// TwinCAT 3 PLC project plc_kfe_vac
// Title: plc_kfe_vac
// Company: SLAC
// ProjectVersion: 0.0.0
// ProgramVersion: 3.1.4022.4
// libraries:
//   LCLS General, * (SLAC)
//   LCLS Vacuum, * (SLAC - LCLS)
//   PMPS, * (SLAC - LCLS)
//   Tc2_Standard, * (Beckhoff Automation GmbH)
//   Tc2_System, * (Beckhoff Automation GmbH)
//   Tc2_Utilities, * (Beckhoff Automation GmbH)
//   Tc3_Module, * (Beckhoff Automation GmbH)
// project tree:
//   DUTs/ ST_EXT_GCC.TcDUT, ST_EXT_ILK.TcDUT
//   / FSV_task.TcTTO, PlcTask.TcTTO
//   GVLs/ GVL_SXR_VAC.TcGVL, GVL_VAC_INTF.TcGVL, GVL_Variables.TcGVL, GVL_VFS.TcGVL
//   POUs/ FB_EXT_TREATY_GAUGE.TcPOU, FB_EXT_TREATY_VGC.TcPOU, FB_EXT_ILK.TcPOU, MAIN.TcPOU, PRG_DIAGNOSTIC.TcPOU, PRG_PMPS.TcPOU, PRG_SXR_VAC.TcPOU, PRG_VAC_INTF.TcPOU, PRG_VFS.TcPOU
// real-time tasks:
//   TASK PlcTask: cycle T#10ms, priority 20, ADS port 350
//   TASK SimTask: cycle T#10ms, priority 21, ADS port 351
//   TASK FSV_task: cycle T#1ms, priority 13, ADS port 352
// I/O:
//   DEVICE Device 1 (EtherCAT), AmsNetId 172.21.92.61.4.1
//     =+-EK1200_00_00 [EK1200-5000 EtherCAT Power supply (2A E-Bus)]
//       =+-ES3064_00_01 [EL3064 4Ch. Ana. Input 0-10V]
//       =+-ES1004_00_02 [EL1004 4Ch. Dig. Input 24V, 3ms]
//       =+-EL2794_00_03 [EL2794 4Ch. Dig. Output 24V AC/DC, 2A, short-circuit-proof]
//       =+-ES3064_00_04 [EL3064 4Ch. Ana. Input 0-10V]
//       =+-ES1004_00_05 [EL1004 4Ch. Dig. Input 24V, 3ms]
//       =+-EL2794_00_06 [EL2794 4Ch. Dig. Output 24V AC/DC, 2A, short-circuit-proof]
//       =+-EL9410_00_07 [EL9410 E-Bus Power Supplier  (Diagnostics)]
//       =+-ES3064_00_08 [EL3064 4Ch. Ana. Input 0-10V]
//       =+-ES1004_00_09 [EL1004 4Ch. Dig. Input 24V, 3ms]
//       =+-EL2794_00_10 [EL2794 4Ch. Dig. Output 24V AC/DC, 2A, short-circuit-proof]
//       =+-ES3064_00_11 [EL3064 4Ch. Ana. Input 0-10V]
//       =+-ES1004_00_12 [EL1004 4Ch. Dig. Input 24V, 3ms]
//       =+-EL2794_00_13 [EL2794 4Ch. Dig. Output 24V AC/DC, 2A, short-circuit-proof]
//       Term 81 (EL6070) [EL6070 1Ch. Licensing-Terminal]
//       =+-EK1110_00_14 [EK1110 EtherCAT extension]
//     =+-EK1100_01_00 [EK1100 EtherCAT Coupler (2A E-Bus)]
//       =+-ES3068_01_01 [EL3068 8Ch. Ana. Input 0-10V]
//       =+-EL2798_01_02 [EL2798 8Ch. Dig. Output 24V AC/DC, 2A, potential-free]
//       =+-ES9187_01_03 [EL9187 Potential Connection, 8 x Ground]
//       =+-ES3068_01_04 [EL3068 8Ch. Ana. Input 0-10V]
//       =+-ES3068_01_05 [EL3068 8Ch. Ana. Input 0-10V]
//       =+-EL2798_01_06 [EL2798 8Ch. Dig. Output 24V AC/DC, 2A, potential-free]
//       =+-ES9187_01_07 [EL9187 Potential Connection, 8 x Ground]
//       =+-ES3068_01_08 [EL3068 8Ch. Ana. Input 0-10V]
//       =+-EL9410_01_09 [EL9410 E-Bus Power Supplier  (Diagnostics)]
//       =+-EL2022_01_10 [EL2022 2Ch. Dig. Output 24V, 2A] (disabled)
//       PMPS_FFO (EL2202) [EL2202 2Ch. Dig. Output 24V, 0.5A]
//       PMPS_PRE [EL6692 EtherCAT Bridge terminal (Primary)]
//       =+-EL6695_01_11 [EL6695 EtherCAT Bridge terminal (Primary)] (disabled)
//       Term 73 (EK1122) [EK1122 2 port EtherCAT junction]
//       =+-EL6695_01_12 [EL6695 EtherCAT Bridge terminal (Primary)] (disabled)
//       Term 74 (EK1122) [EK1122 2 port EtherCAT junction]
//       =+-EL6695_01_13 [EL6695 EtherCAT Bridge terminal (Primary)] (disabled)
//       Term 75 (EK1122) [EK1122 2 port EtherCAT junction]
//       =+-EL6695_01_14 [EL6695 EtherCAT Bridge terminal (Primary)] (disabled)
//       Term 76 (EL9011) [EL9011 End Terminal]
//     =+-EK1100_02_00 [EK1100 EtherCAT Coupler (2A E-Bus)]
//       =+-EL3064_02_01 [EL3064 4Ch. Ana. Input 0-10V]
//       =+-EL9070_02_02 [EL9070 Shield terminal]
//       =+-ES1008_02_03 [EL1008 8Ch. Dig. Input 24V, 3ms]
//       =+-ES9184_02_04 [EL9184 Potential Connection, 8 x 24V, 8 x Ground]
//       =+-ES2008_02_05 [EL2008 8Ch. Dig. Output 24V, 0.5A]
//       =+-EL2798_02_06 [EL2798 8Ch. Dig. Output 24V AC/DC, 2A, potential-free]
//       =+-EL3064_02_07 [EL3064 4Ch. Ana. Input 0-10V]
//       =+-EL2794_02_08 [EL2794 4Ch. Dig. Output 24V AC/DC, 2A, short-circuit-proof]
//       =+-EL1004_02_09 [EL1004 4Ch. Dig. Input 24V, 3ms]
//       =+-EL9505_02_10 [EL9505 Power supply terminal 5V]
//       =+-EL1124_02_11 [EL1124 4Ch. Dig. Input 5V, 10µs, Sensor Power]
//       =+-EL9011_02_12 [EL9011 End Terminal]
//     =+-EK1100_03_00 [EK1100 EtherCAT Coupler (2A E-Bus)]
//       =+-ES1004_03_01 [EL1004 4Ch. Dig. Input 24V, 3ms]
//       =+-ES2004_03_02 [EL2004 4Ch. Dig. Output 24V, 0.5A]
//       =+-ES2004_03_03 [EL2004 4Ch. Dig. Output 24V, 0.5A]
//       =+-EL1004_03_04 [EL1004 4Ch. Dig. Input 24V, 3ms]
//       =+-EL3064_03_05 [EL3064 4Ch. Ana. Input 0-10V]
//       =+-EL9070_03_06 [EL9070 Shield terminal]
//       =+-ES1008_03_07 [EL1008 8Ch. Dig. Input 24V, 3ms]
//       =+-ES9184_03_08 [EL9184 Potential Connection, 8 x 24V, 8 x Ground]
//       =+-ES2008_03_09 [EL2008 8Ch. Dig. Output 24V, 0.5A]
//       =+-EL2798_03_10 [EL2798 8Ch. Dig. Output 24V AC/DC, 2A, potential-free]
//       =+-EL9011_03_11 [EL9011 End Terminal]
//     =+-EP2338_04_00 [EP2338-0002 8 Ch. Dig. Input/Output 24V, 0,5A, M12]
//     =+-EP2338_05_00 [EP2338-0002 8 Ch. Dig. Input/Output 24V, 0,5A, M12]
//     =+-EK1100_05_01 [EK1100 EtherCAT Coupler (2A E-Bus)]
//       =+-ES1004_05_02 [EL1004 4Ch. Dig. Input 24V, 3ms]
//       =+-ES2202_05_03 [EL2202 2Ch. Dig. Output 24V, 0.5A]
//       =+-ES2202_05_04 [EL2202 2Ch. Dig. Output 24V, 0.5A]
//       Term 55 (EL9011) [EL9011 End Terminal]
//     =+-EP2338_06_00 [EP2338-0002 8 Ch. Dig. Input/Output 24V, 0,5A, M12]
//     =+-EP2338_07_00 [EP2338-0002 8 Ch. Dig. Input/Output 24V, 0,5A, M12]
//     =+-EP3174_07_01 [EP3174-0002 4Ch. Ana. Input +/-10V, 0-10V, 0/4-20mA configurable]
//     =+-EP2624_07_02 [EP2624-0002 4Ch. Relay Output, NO (125V AC / 30V DC)]
//     =+-EP2338_08_00 [EP2338-0002 8 Ch. Dig. Input/Output 24V, 0,5A, M12]
//     =+-EP3174_08_01 [EP3174-0002 4Ch. Ana. Input +/-10V, 0-10V, 0/4-20mA configurable]
//     =+-EP2624_08_02 [EP2624-0002 4Ch. Relay Output, NO (125V AC / 30V DC)]
//     =+-EP3174_09_00 [EP3174-0002 4Ch. Ana. Input +/-10V, 0-10V, 0/4-20mA configurable]
//     =+-EP2624_09_01 [EP2624-0002 4Ch. Relay Output, NO (125V AC / 30V DC)]
//     =+-EP2338_09_02 [EP2338-0002 8 Ch. Dig. Input/Output 24V, 0,5A, M12]
//     =+-EP2338_09_03 [EP2338-0002 8 Ch. Dig. Input/Output 24V, 0,5A, M12]
//     =+-EP3174_10_00 [EP3174-0002 4Ch. Ana. Input +/-10V, 0-10V, 0/4-20mA configurable]
//     =+-EP2624_10_01 [EP2624-0002 4Ch. Relay Output, NO (125V AC / 30V DC)]
//     =+-EP2338_10_02 [EP2338-0002 8 Ch. Dig. Input/Output 24V, 0,5A, M12]
//   DEVICE SimDevice 2 (EtherCAT Simulation) (disabled), AmsNetId 10.0.1.49.3.1
//     =+-ES3064_00_01 // EL3064-0000-0020
//     =+-ES1004_00_02 // EL1004-0000-0019
//     =+-EL2794_00_03 // EL2794-0000-0016
//     =+-ES3064_00_04 // EL3064-0000-0020
//     =+-ES1004_00_05 // EL1004-0000-0019
//     =+-EL2794_00_06 // EL2794-0000-0016
//     =+-EL9410_00_07 // EL9410-0000-0017
//     =+-ES3064_00_08 // EL3064-0000-0020
//     =+-ES1004_00_09 // EL1004-0000-0019
//     =+-EL2794_00_10 // EL2794-0000-0016
//     =+-ES3064_00_11 // EL3064-0000-0020
//     =+-ES1004_00_12 // EL1004-0000-0019
//     =+-EL2794_00_13 // EL2794-0000-0016
//     =+-EK1110_00_14 // EK1110-0000-0017
//     =+-EK1100_01_00 // EK1100-0000-0018
//     =+-ES3068_01_01 // EL3068-0000-0020
//     =+-EL2798_01_02 // EL2798-0000-0018
//     =+-ES3068_01_04 // EL3068-0000-0020
//     =+-ES3068_01_05 // EL3068-0000-0020
//     =+-EL2798_01_06 // EL2798-0000-0018
//     =+-ES3068_01_08 // EL3068-0000-0020
//     =+-EL9410_01_09 // EL9410-0000-0017
//     =+-EL2202_01_10 // EL2022-0000-0018
//     =+-EL6695_01_11 // EL6695-0000-0005
//     =+-EL6695_01_12 // EL6695-0000-0005
//     =+-EL6695_01_13 // EL6695-0000-0005
//     =+-EL6695_01_14 // EL6695-0000-0005
//     =+-EK1100_02_00 // EK1100-0000-0018
//     =+-EL3064_02_01 // EL3064-0000-0020
//     =+-ES1008_02_03 // EL1008-0000-0018
//     =+-ES2008_02_05 // EL2008-0000-0018
//     =+-EL2798_02_06 // EL2798-0000-0018
//     =+-EK1100_03_00 // EK1100-0000-0018
//     =+-ES1004_03_01 // EL1004-0000-0019
//     =+-ES2004_03_02 // EL2004-0000-0018
//     =+-ES2004_03_03 // EL2004-0000-0018
//     =+-ES1004_03_04 // EL1008-0000-0018
//     =+-EL3064_03_05 // EL3064-0000-0020
//     =+-ES1008_03_07 // EL1008-0000-0018
//     =+-ES2008_03_09 // EL2008-0000-0018
//     =+-EL2798_03_10 // EL2798-0000-0018
//     =+-EP2338_04_00 // EP2338-0002-0023
//     =+-EP2338_05_00 // EP2338-0002-0023
//     =+-EK1100_05_01 // EK1100-0000-0018
//     =+-ES1004_05_02 // EL1004-0000-0019
//     =+-ES2202_05_03 // EL2202-0000-0019
//     =+-ES2202_05_04 // EL2202-0000-0019
//     =+-ES9505_05_05 // EL9505-0000-0018
//     =+-ES1124_05_06 // EL1124-0000-0018
//     =+-EP2338_06_00 // EP2338-0002-0023
//     =+-EP2338_07_00 // EP2338-0002-0023
//     =+-EP3174_07_01 // EP3174-0002-0023
//     =+-EP2624_07_02 // EP2624-0002-0019
//     =+-EP2338_08_00 // EP2338-0002-0023
//     =+-EP3174_08_01 // EP3174-0002-0023
//     =+-EP2624_08_02 // EP2624-0002-0019
//     =+-EP3174_09_00 // EP3174-0002-0023
//     =+-EP2624_09_01 // EP2624-0002-0019
//     =+-EP2338_09_02 // EP2338-0002-0023
//     =+-EP2338_09_03 // EP2338-0002-0023
//     =+-EP3174_10_00 // EP3174-0002-0023
//     =+-EP2624_10_01 // EP2624-0002-0019
//     =+-EP2338_10_02 // EP2338-0002-0023
//     =+-EP3174_11_00 // EP3174-0002-0023
//     =+-EP2624_11_01 // EP2624-0002-0019
//     =+-EP2338_11_02 // EP2338-0002-0023
//     =+-EK1100_11_03 // EK1100-0000-0018
//     =+-ES1004_11_04 // EL1004-0000-0019
//     =+-ES2202_11_05 // EL2202-0000-0019
//     =+-ES2202_11_06 // EL2202-0000-0019
//     =+-ES9505_11_07 // EL9505-0000-0018
//     =+-ES1124_11_08 // EL1124-0000-0018
//     =+-EP3174_12_00 // EP3174-0002-0023
//     =+-EP2624_12_01 // EP2624-0002-0019
//     =+-EP3174_13_00 // EP3174-0002-0023
//     =+-EP2624_13_01 // EP2624-0002-0019
//     =+-EP2338_14_00 // EP2338-0002-0023
//     =+-EP3174_14_01 // EP3174-0002-0023
//     =+-EP2624_14_02 // EP2624-0002-0019
//     =+-EK1100_15_00 // EK1100-0000-0018
//     =+-ES3064_15_01 // EL3064-0000-0020
//     =+-ES1004_15_02 // EL1004-0000-0019
//     =+-EL2794_15_03 // EL2794-0000-0016
//     =+-ES3064_15_04 // EL3064-0000-0020
//     =+-ES1004_15_05 // EL1004-0000-0019
//     =+-EL2794_15_06 // EL2794-0000-0016
// variable links:
//   plc_kfe_vac/plc_kfe_vac Instance <-> Device 1 (EtherCAT)
//     PlcTask Inputs/GVL_Variables.fbEcatDiagWrapper.arrEcMasterNetId <-> InfoData/AmsNetId
//     PlcTask Inputs/GVL_Variables.fbEcatDiagWrapper.nEcMasterDevState <-> Inputs/DevState
//     PlcTask Inputs/GVL_Variables.fbEcatDiagWrapper.nEcMasterDeviceId <-> InfoData/DevId
//     PlcTask Inputs/GVL_Variables.fbEcatDiagWrapper.nEcMasterSlaveCount <-> Inputs/SlaveCount
//     PlcTask Inputs/GVL_Variables.fbEcatDiagWrapper.nEcMasterSlaveCountCfg <-> InfoData/CfgSlaveCount
//     PlcTask Inputs/GVL_Variables.fbEcatDiagWrapper.wFrmXWcState <-> Inputs/Frm1WcState
//   plc_kfe_vac/plc_kfe_vac Instance <-> Device 1 (EtherCAT)/=+-EK1100_01_00/=+-EL2798_01_02
//     PlcTask Outputs/GVL_SXR_VAC.fb_IM1K0_XTES_GCC_1.q_xHV_DIS <-> Channel 2/GVL_SXR_VAC.fb_IM1K0_XTES_GCC_1.q_xHV_DIS
//     PlcTask Outputs/GVL_SXR_VAC.fb_PCPM3B_GFS_1.q_xHV_DIS <-> Channel 5/GVL_SXR_VAC.fb_PCPM3B_GFS_1.q_xHV_DIS
//     PlcTask Outputs/GVL_SXR_VAC.fb_RTDSK0_GCC_1.q_xHV_DIS <-> Channel 1/GVL_SXR_VAC.fb_RTDSK0_GCC_1.q_xHV_DIS
//     PlcTask Outputs/GVL_SXR_VAC.fb_SL1K0_POWER_GCC_1.q_xHV_DIS <-> Channel 4/GVL_SXR_VAC.fb_SL1K0_POWER_GCC_1.q_xHV_DIS
//   plc_kfe_vac/plc_kfe_vac Instance <-> Device 1 (EtherCAT)/=+-EK1100_01_00/=+-EL2798_01_06
//     PlcTask Outputs/GVL_SXR_VAC.fb_PA1K0_GCC_1.q_xHV_DIS <-> Channel 4/GVL_SXR_VAC.fb_PA1K0_GCC_1.q_xHV_DIS
//     PlcTask Outputs/GVL_SXR_VAC.fb_TV2K0_GCC_1.q_xHV_DIS <-> Channel 1/GVL_SXR_VAC.fb_TV2K0_GCC_1.q_xHV_DIS
//     PlcTask Outputs/GVL_SXR_VAC.fb_TV2K0_GCC_2.q_xHV_DIS <-> Channel 2/GVL_SXR_VAC.fb_TV2K0_GCC_2.q_xHV_DIS
//   plc_kfe_vac/plc_kfe_vac Instance <-> Device 1 (EtherCAT)/=+-EK1100_01_00/=+-ES3068_01_01
//     PlcTask Inputs/GVL_SXR_VAC.fb_IM1K0_XTES_GCC_1.i_iPRESS_R <-> AI Standard Channel 3/GVL_SXR_VAC.fb_IM1K0_XTES_GCC_1.i_iPRESS_R
//     PlcTask Inputs/GVL_SXR_VAC.fb_IM1K0_XTES_GPI_1.i_iPRESS_R <-> AI Standard Channel 6/GVL_SXR_VAC.fb_IM1K0_XTES_GPI_1.i_iPRESS_R
//     PlcTask Inputs/GVL_SXR_VAC.fb_RTDSK0_GCC_1.i_iPRESS_R <-> AI Standard Channel 1/GVL_SXR_VAC.fb_RTDSK0_GCC_1.i_iPRESS_R
//     PlcTask Inputs/GVL_SXR_VAC.fb_RTDSK0_GPI_1.i_iPRESS_R <-> AI Standard Channel 5/GVL_SXR_VAC.fb_RTDSK0_GPI_1.i_iPRESS_R
//   plc_kfe_vac/plc_kfe_vac Instance <-> Device 1 (EtherCAT)/=+-EK1100_01_00/=+-ES3068_01_04
//     PlcTask Inputs/GVL_SXR_VAC.fb_PCPM3B_GFS_1.i_iPRESS_R <-> AI Standard Channel 3/GVL_SXR_VAC.fb_PCPM3B_GFS_1.i_iPRESS_R
//     PlcTask Inputs/GVL_SXR_VAC.fb_SL1K0_POWER_GCC_1.i_iPRESS_R <-> AI Standard Channel 1/GVL_SXR_VAC.fb_SL1K0_POWER_GCC_1.i_iPRESS_R
//     PlcTask Inputs/GVL_SXR_VAC.fb_SL1K0_POWER_GPI_1.i_iPRESS_R <-> AI Standard Channel 5/GVL_SXR_VAC.fb_SL1K0_POWER_GPI_1.i_iPRESS_R
//   plc_kfe_vac/plc_kfe_vac Instance <-> Device 1 (EtherCAT)/=+-EK1100_01_00/=+-ES3068_01_05
//     PlcTask Inputs/GVL_SXR_VAC.fb_TV2K0_GCC_1.i_iPRESS_R <-> AI Standard Channel 1/GVL_SXR_VAC.fb_TV2K0_GCC_1.i_iPRESS_R
//     PlcTask Inputs/GVL_SXR_VAC.fb_TV2K0_GCC_2.i_iPRESS_R <-> AI Standard Channel 3/GVL_SXR_VAC.fb_TV2K0_GCC_2.i_iPRESS_R
//     PlcTask Inputs/GVL_SXR_VAC.fb_TV2K0_GPI_1.i_iPRESS_R <-> AI Standard Channel 5/GVL_SXR_VAC.fb_TV2K0_GPI_1.i_iPRESS_R
//     PlcTask Inputs/GVL_SXR_VAC.fb_TV2K0_GPI_2.i_iPRESS_R <-> AI Standard Channel 6/GVL_SXR_VAC.fb_TV2K0_GPI_2.i_iPRESS_R
//   plc_kfe_vac/plc_kfe_vac Instance <-> Device 1 (EtherCAT)/=+-EK1100_01_00/=+-ES3068_01_08
//     PlcTask Inputs/GVL_SXR_VAC.fb_PA1K0_GCC_1.i_iPRESS_R <-> AI Standard Channel 1/GVL_SXR_VAC.fb_PA1K0_GCC_1.i_iPRESS_R
//     PlcTask Inputs/GVL_SXR_VAC.fb_PA1K0_GPI_1.i_iPRESS_R <-> AI Standard Channel 5/GVL_SXR_VAC.fb_PA1K0_GPI_1.i_iPRESS_R
//   plc_kfe_vac/plc_kfe_vac Instance <-> Device 1 (EtherCAT)/=+-EK1100_01_00/PMPS_FFO (EL2202)
//     FSV_task Outputs/GVL_Variables.g_FastFaultOutput2.q_xFastFaultOut <-> Channel 2/Output
//     PlcTask Outputs/GVL_Variables.g_FastFaultOutputAll.q_xFastFaultOut <-> Channel 1/Output
//   plc_kfe_vac/plc_kfe_vac Instance <-> Device 1 (EtherCAT)/=+-EK1100_01_00/PMPS_PRE
//     PlcTask Inputs/PRG_PMPS.fbArbiterIO.i_stCurrentBP <-> IO Inputs/CurrentBP
//     PlcTask Inputs/PRG_PMPS.fbArbiterIO.xTxPDO_state <-> SYNC Inputs/TxPDO state
//     PlcTask Inputs/PRG_PMPS.fbArbiterIO.xTxPDO_toggle <-> SYNC Inputs/TxPDO toggle
//     PlcTask Outputs/PRG_PMPS.fbArbiterIO.q_stRequestedBP <-> IO Outputs/RequestedBP
//   plc_kfe_vac/plc_kfe_vac Instance <-> Device 1 (EtherCAT)/=+-EK1100_02_00/=+-EL1004_02_09
//     PlcTask Inputs/GVL_SXR_VAC.fb_SL1K0_PIP_1.i_xSP_DI <-> Channel 1/Input
//   plc_kfe_vac/plc_kfe_vac Instance <-> Device 1 (EtherCAT)/=+-EK1100_02_00/=+-EL1124_02_11
//     FSV_task Inputs/GVL_VFS.fb_TV2K0_VFS_1.i_xTrigger <-> Channel 1/GVL_SXR_VAC_FS_DEVICES.fb_TV2K0_VFS_1.i_xTrigger
//   plc_kfe_vac/plc_kfe_vac Instance <-> Device 1 (EtherCAT)/=+-EK1100_02_00/=+-EL2794_02_08
//     PlcTask Outputs/GVL_SXR_VAC.fb_SL1K0_PIP_1.q_xHVEna_DO <-> Channel 1/Output
//   plc_kfe_vac/plc_kfe_vac Instance <-> Device 1 (EtherCAT)/=+-EK1100_02_00/=+-EL2798_02_06
//     PlcTask Outputs/GVL_VAC_INTF.fb_TMO_ILK_Lower.q_xILK_OK_DO <-> Channel 2/Output
//     PlcTask Outputs/GVL_VAC_INTF.fb_TMO_ILK_Uppper.q_xILK_OK_DO <-> Channel 1/Output
//   plc_kfe_vac/plc_kfe_vac Instance <-> Device 1 (EtherCAT)/=+-EK1100_02_00/=+-EL3064_02_07
//     PlcTask Inputs/GVL_SXR_VAC.fb_SL1K0_PIP_1.i_iPRESS <-> AI Standard Channel 1/Value
//   plc_kfe_vac/plc_kfe_vac Instance <-> Device 1 (EtherCAT)/=+-EK1100_02_00/=+-ES1008_02_03
//     PlcTask Inputs/GVL_VAC_INTF.fb_PC1K1_INTF_GCC_1.i_xEXT_Press_OK <-> Channel 1/GVL_VAC_INTF.fb_PC1K1_INTF_GCC_1.i_xEXT_Press_OK
//     PlcTask Inputs/GVL_VAC_INTF.fb_PC1K3_INTF_PIP_1.i_xEXT_Press_OK <-> Channel 3/Input
//   plc_kfe_vac/plc_kfe_vac Instance <-> Device 1 (EtherCAT)/=+-EK1100_03_00/=+-EL1004_03_04
//     PlcTask Inputs/GVL_SXR_VAC.fb_AT1K0_GAS_VGC_1.i_xClsLS <-> Channel 2/Input
//     PlcTask Inputs/GVL_SXR_VAC.fb_AT1K0_GAS_VGC_1.i_xOpnLS <-> Channel 1/Input
//     PlcTask Inputs/GVL_SXR_VAC.fb_IM1K0_XTES_VGC_1.i_xClsLS <-> Channel 4/Input
//     PlcTask Inputs/GVL_SXR_VAC.fb_IM1K0_XTES_VGC_1.i_xOpnLS <-> Channel 3/Input
//   plc_kfe_vac/plc_kfe_vac Instance <-> Device 1 (EtherCAT)/=+-EK1100_03_00/=+-ES1004_03_01
//     PlcTask Inputs/GVL_SXR_VAC.fb_EM1K0_GMD_VGC_1.i_xClsLS <-> Channel 4/GVL_SXR_VAC.fb_EM1K0_GMD_VGC_1.i_xClsLS
//     PlcTask Inputs/GVL_SXR_VAC.fb_EM1K0_GMD_VGC_1.i_xOpnLS <-> Channel 3/GVL_SXR_VAC.fb_EM1K0_GMD_VGC_1.i_xOpnLS
//     PlcTask Inputs/GVL_SXR_VAC.fb_RTDSK0_VGC_1.i_xClsLS <-> Channel 2/GVL_SXR_VAC.fb_RTDSK0_VGC_1.i_xClsLS
//     PlcTask Inputs/GVL_SXR_VAC.fb_RTDSK0_VGC_1.i_xOpnLS <-> Channel 1/GVL_SXR_VAC.fb_RTDSK0_VGC_1.i_xOpnLS
//   plc_kfe_vac/plc_kfe_vac Instance <-> Device 1 (EtherCAT)/=+-EK1100_03_00/=+-ES1008_03_07
//     PlcTask Inputs/GVL_VAC_INTF.fb_TV1K0_INTF_GCC_1.i_xEXT_Press_OK <-> Channel 3/GVL_VAC_INTF.fb_TV1K0_INTF_GCC_1.i_xEXT_Press_OK
//   plc_kfe_vac/plc_kfe_vac Instance <-> Device 1 (EtherCAT)/=+-EK1100_03_00/=+-ES2004_03_02
//     PlcTask Outputs/GVL_SXR_VAC.fb_EM1K0_GMD_VGC_1.q_xOPN_DO <-> Channel 3/GVL_SXR_VAC.fb_EM1K0_GMD_VGC_1.q_xOPN_DO
//     PlcTask Outputs/GVL_SXR_VAC.fb_EM1K0_GMD_VGC_1.q_xOPN_DO <-> Channel 4/GVL_SXR_VAC.fb_EM1K0_GMD_VGC_1.q_xOPN_DO
//     PlcTask Outputs/GVL_SXR_VAC.fb_RTDSK0_VGC_1.q_xOPN_DO <-> Channel 1/GVL_SXR_VAC.fb_RTDSK0_VGC_1.q_xOPN_DO
//     PlcTask Outputs/GVL_SXR_VAC.fb_RTDSK0_VGC_1.q_xOPN_DO <-> Channel 2/GVL_SXR_VAC.fb_RTDSK0_VGC_1.q_xOPN_DO
//   plc_kfe_vac/plc_kfe_vac Instance <-> Device 1 (EtherCAT)/=+-EK1100_03_00/=+-ES2004_03_03
//     PlcTask Outputs/GVL_SXR_VAC.fb_AT1K0_GAS_VGC_1.q_xOPN_DO <-> Channel 1/GVL_SXR_VAC.fb_AT1K0_GAS_VGC_1.q_xOPN_DO
//     PlcTask Outputs/GVL_SXR_VAC.fb_AT1K0_GAS_VGC_1.q_xOPN_DO <-> Channel 2/GVL_SXR_VAC.fb_AT1K0_GAS_VGC_1.q_xOPN_DO
//     PlcTask Outputs/GVL_SXR_VAC.fb_IM1K0_XTES_VGC_1.q_xOPN_DO <-> Channel 3/Output
//     PlcTask Outputs/GVL_SXR_VAC.fb_IM1K0_XTES_VGC_1.q_xOPN_DO <-> Channel 4/Output
//   plc_kfe_vac/plc_kfe_vac Instance <-> Device 1 (EtherCAT)/=+-EK1100_05_01/=+-ES1004_05_02
//     FSV_task Inputs/GVL_VFS.fb_TV2K0_VFS_1.i_xClsLS <-> Channel 1/GVL_SXR_VAC_FS_DEVICES.fb_TV2K0_VFS_1.i_xClsLS
//     FSV_task Inputs/GVL_VFS.fb_TV2K0_VFS_1.i_xOpnLS <-> Channel 2/GVL_SXR_VAC_FS_DEVICES.fb_TV2K0_VFS_1.i_xOpnLS
//   plc_kfe_vac/plc_kfe_vac Instance <-> Device 1 (EtherCAT)/=+-EK1100_05_01/=+-ES2202_05_03
//     FSV_task Outputs/GVL_VFS.fb_TV2K0_VFS_1.q_xClose_A <-> Channel 1/GVL_SXR_VAC_FS_DEVICES.fb_TV2K0_VFS_1.q_xClose_A
//     FSV_task Outputs/GVL_VFS.fb_TV2K0_VFS_1.q_xClose_B <-> Channel 2/GVL_SXR_VAC_FS_DEVICES.fb_TV2K0_VFS_1.q_xClose_B
//   plc_kfe_vac/plc_kfe_vac Instance <-> Device 1 (EtherCAT)/=+-EK1100_05_01/=+-ES2202_05_04
//     FSV_task Outputs/GVL_VFS.fb_TV2K0_VFS_1.q_xClose_C <-> Channel 1/GVL_SXR_VAC_FS_DEVICES.fb_TV2K0_VFS_1.q_xClose_C
//     FSV_task Outputs/GVL_VFS.fb_TV2K0_VFS_1.q_xOPN_DO <-> Channel 2/GVL_SXR_VAC_FS_DEVICES.fb_TV2K0_VFS_1.q_xOPN_DO
//   plc_kfe_vac/plc_kfe_vac Instance <-> Device 1 (EtherCAT)/=+-EK1200_00_00/=+-EL2794_00_03
//     PlcTask Outputs/GVL_SXR_VAC.fb_RTDSK0_PIP_{1..4}.q_xHVEna_DO <-> Channel {1..4}/GVL_SXR_VAC.fb_RTDSK0_PIP_{1..4}.q_xHVEna_DO  (4 links)
//   plc_kfe_vac/plc_kfe_vac Instance <-> Device 1 (EtherCAT)/=+-EK1200_00_00/=+-EL2794_00_06
//     PlcTask Outputs/GVL_SXR_VAC.fb_MR1K1_BEND_PIP_1.q_xHVEna_DO <-> Channel 3/GVL_SXR_VAC.fb_MR1K1_BEND_PIP_1.q_xHVEna_DO
//     PlcTask Outputs/GVL_SXR_VAC.fb_MR1K3_TXI_PIP_1.q_xHVEna_DO <-> Channel 4/GVL_SXR_VAC.fb_MR1K3_TXI_PIP_1.q_xHVEna_DO
//     PlcTask Outputs/GVL_SXR_VAC.fb_RTDSK0_PIP_5.q_xHVEna_DO <-> Channel 2/GVL_SXR_VAC.fb_RTDSK0_PIP_5.q_xHVEna_DO
//   plc_kfe_vac/plc_kfe_vac Instance <-> Device 1 (EtherCAT)/=+-EK1200_00_00/=+-EL2794_00_10
//     PlcTask Outputs/GVL_SXR_VAC.fb_MR2K3_TXI_PIP_1.q_xHVEna_DO <-> Channel 1/GVL_SXR_VAC.fb_MR2K3_TXI_PIP_1.q_xHVEna_DO
//     PlcTask Outputs/GVL_SXR_VAC.fb_SP1K1_MONO_PIP_1.q_xHVEna_DO <-> Channel 2/GVL_SXR_VAC.fb_SP1K1_MONO_PIP_1.q_xHVEna_DO
//     PlcTask Outputs/GVL_SXR_VAC.fb_SP1K1_MONO_PIP_2.q_xHVEna_DO <-> Channel 3/GVL_SXR_VAC.fb_SP1K1_MONO_PIP_2.q_xHVEna_DO
//     PlcTask Outputs/GVL_SXR_VAC.fb_TV3K0_PIP_1.q_xHVEna_DO <-> Channel 4/GVL_SXR_VAC.fb_TV3K0_PIP_1.q_xHVEna_DO
//   plc_kfe_vac/plc_kfe_vac Instance <-> Device 1 (EtherCAT)/=+-EK1200_00_00/=+-EL2794_00_13
//     PlcTask Outputs/GVL_SXR_VAC.fb_PA1K0.q_xHVEna_DO <-> Channel 2/GVL_SXR_VAC.fb_PA1K0.q_xHVEna_DO
//     PlcTask Outputs/GVL_SXR_VAC.fb_PA1K0_PIP_1.q_xHVEna_DO <-> Channel 3/GVL_SXR_VAC.fb_PA1K0_PIP_1.q_xHVEna_DO
//     PlcTask Outputs/GVL_SXR_VAC.fb_PCPM3B_PIP_1.q_xHVEna_DO <-> Channel 1/GVL_SXR_VAC.fb_PCPM3B_PIP_1.q_xHVEna_DO
//   plc_kfe_vac/plc_kfe_vac Instance <-> Device 1 (EtherCAT)/=+-EK1200_00_00/=+-ES1004_00_02
//     PlcTask Inputs/GVL_SXR_VAC.fb_RTDSK0_PIP_{1..4}.i_xSP_DI <-> Channel {1..4}/GVL_SXR_VAC.fb_RTDSK0_PIP_{1..4}.i_xSP_DI  (4 links)
//   plc_kfe_vac/plc_kfe_vac Instance <-> Device 1 (EtherCAT)/=+-EK1200_00_00/=+-ES1004_00_05
//     PlcTask Inputs/GVL_SXR_VAC.fb_MR1K1_BEND_PIP_1.i_xSP_DI <-> Channel 3/GVL_SXR_VAC.fb_MR1K1_BEND_PIP_1.i_xSP_DI
//     PlcTask Inputs/GVL_SXR_VAC.fb_MR1K3_TXI_PIP_1.i_xSP_DI <-> Channel 4/GVL_SXR_VAC.fb_MR1K3_TXI_PIP_1.i_xSP_DI
//     PlcTask Inputs/GVL_SXR_VAC.fb_RTDSK0_PIP_5.i_xSP_DI <-> Channel 2/GVL_SXR_VAC.fb_RTDSK0_PIP_5.i_xSP_DI
//   plc_kfe_vac/plc_kfe_vac Instance <-> Device 1 (EtherCAT)/=+-EK1200_00_00/=+-ES1004_00_09
//     PlcTask Inputs/GVL_SXR_VAC.fb_MR2K3_TXI_PIP_1.i_xSP_DI <-> Channel 1/GVL_SXR_VAC.fb_MR2K3_TXI_PIP_1.i_xSP_DI
//     PlcTask Inputs/GVL_SXR_VAC.fb_SP1K1_MONO_PIP_1.i_xSP_DI <-> Channel 2/GVL_SXR_VAC.fb_SP1K1_MONO_PIP_1.i_xSP_DI
//     PlcTask Inputs/GVL_SXR_VAC.fb_SP1K1_MONO_PIP_2.i_xSP_DI <-> Channel 3/GVL_SXR_VAC.fb_SP1K1_MONO_PIP_2.i_xSP_DI
//     PlcTask Inputs/GVL_SXR_VAC.fb_TV3K0_PIP_1.i_xSP_DI <-> Channel 4/GVL_SXR_VAC.fb_TV3K0_PIP_1.i_xSP_DI
//   plc_kfe_vac/plc_kfe_vac Instance <-> Device 1 (EtherCAT)/=+-EK1200_00_00/=+-ES1004_00_12
//     PlcTask Inputs/GVL_SXR_VAC.fb_PA1K0.i_xSP_DI <-> Channel 2/GVL_SXR_VAC.fb_PA1K0.i_xSP_DI
//     PlcTask Inputs/GVL_SXR_VAC.fb_PA1K0_PIP_1.i_xSP_DI <-> Channel 3/GVL_SXR_VAC.fb_PA1K0_PIP_1.i_xSP_DI
//     PlcTask Inputs/GVL_SXR_VAC.fb_PCPM3B_PIP_1.i_xSP_DI <-> Channel 1/GVL_SXR_VAC.fb_PCPM3B_PIP_1.i_xSP_DI
//   plc_kfe_vac/plc_kfe_vac Instance <-> Device 1 (EtherCAT)/=+-EK1200_00_00/=+-ES3064_00_01
//     PlcTask Inputs/GVL_SXR_VAC.fb_RTDSK0_PIP_{1..4}.i_iPRESS <-> AI Standard Channel {1..4}/GVL_SXR_VAC.fb_RTDSK0_PIP_{1..4}.i_iPRESS  (4 links)
//   plc_kfe_vac/plc_kfe_vac Instance <-> Device 1 (EtherCAT)/=+-EK1200_00_00/=+-ES3064_00_04
//     PlcTask Inputs/GVL_SXR_VAC.fb_MR1K1_BEND_PIP_1.i_iPRESS <-> AI Standard Channel 3/GVL_SXR_VAC.fb_MR1K1_BEND_PIP_1.i_iPRESS
//     PlcTask Inputs/GVL_SXR_VAC.fb_MR1K3_TXI_PIP_1.i_iPRESS <-> AI Standard Channel 4/GVL_SXR_VAC.fb_MR1K3_TXI_PIP_1.i_iPRESS
//     PlcTask Inputs/GVL_SXR_VAC.fb_RTDSK0_PIP_5.i_iPRESS <-> AI Standard Channel 2/GVL_SXR_VAC.fb_RTDSK0_PIP_5.i_iPRESS
//   plc_kfe_vac/plc_kfe_vac Instance <-> Device 1 (EtherCAT)/=+-EK1200_00_00/=+-ES3064_00_08
//     PlcTask Inputs/GVL_SXR_VAC.fb_MR2K3_TXI_PIP_1.i_iPRESS <-> AI Standard Channel 1/GVL_SXR_VAC.fb_MR2K3_TXI_PIP_1.i_iPRESS
//     PlcTask Inputs/GVL_SXR_VAC.fb_SP1K1_MONO_PIP_1.i_iPRESS <-> AI Standard Channel 2/GVL_SXR_VAC.fb_SP1K1_MONO_PIP_1.i_iPRESS
//     PlcTask Inputs/GVL_SXR_VAC.fb_SP1K1_MONO_PIP_2.i_iPRESS <-> AI Standard Channel 3/GVL_SXR_VAC.fb_SP1K1_MONO_PIP_2.i_iPRESS
//     PlcTask Inputs/GVL_SXR_VAC.fb_TV3K0_PIP_1.i_iPRESS <-> AI Standard Channel 4/GVL_SXR_VAC.fb_TV3K0_PIP_1.i_iPRESS
//   plc_kfe_vac/plc_kfe_vac Instance <-> Device 1 (EtherCAT)/=+-EK1200_00_00/=+-ES3064_00_11
//     PlcTask Inputs/GVL_SXR_VAC.fb_PA1K0.i_iPRESS <-> AI Standard Channel 2/GVL_SXR_VAC.fb_PA1K0.i_iPRESS
//     PlcTask Inputs/GVL_SXR_VAC.fb_PA1K0_PIP_1.i_iPRESS <-> AI Standard Channel 3/GVL_SXR_VAC.fb_PA1K0_PIP_1.i_iPRESS
//     PlcTask Inputs/GVL_SXR_VAC.fb_PCPM3B_PIP_1.i_iPRESS <-> AI Standard Channel 1/GVL_SXR_VAC.fb_PCPM3B_PIP_1.i_iPRESS
//   plc_kfe_vac/plc_kfe_vac Instance <-> Device 1 (EtherCAT)/=+-EP2338_04_00
//     PlcTask Inputs/GVL_SXR_VAC.fb_EM2K0_XGMD_VGC_1.i_xClsLS <-> Channel 2/GVL_SXR_VAC.fb_EM2K0_XGMD_VGC_1.i_xClsLS
//     PlcTask Inputs/GVL_SXR_VAC.fb_EM2K0_XGMD_VGC_2.i_xClsLS <-> Channel 6/GVL_SXR_VAC.fb_EM2K0_XGMD_VGC_2.i_xClsLS
//     PlcTask Inputs/GVL_SXR_VAC.fb_EM2K0_XGMD_VGC_1.i_xOpnLS <-> Channel 1/GVL_SXR_VAC.fb_EM2K0_XGMD_VGC_1.i_xOpnLS
//     PlcTask Inputs/GVL_SXR_VAC.fb_EM2K0_XGMD_VGC_2.i_xOpnLS <-> Channel 5/GVL_SXR_VAC.fb_EM2K0_XGMD_VGC_2.i_xOpnLS
//     PlcTask Outputs/GVL_SXR_VAC.fb_EM2K0_XGMD_VGC_1.q_xOPN_DO <-> Channel 11/GVL_SXR_VAC.fb_EM2K0_XGMD_VGC_1.q_xOPN_DO
//     PlcTask Outputs/GVL_SXR_VAC.fb_EM2K0_XGMD_VGC_2.q_xOPN_DO <-> Channel 15/GVL_SXR_VAC.fb_EM2K0_XGMD_VGC_2.q_xOPN_DO
//   plc_kfe_vac/plc_kfe_vac Instance <-> Device 1 (EtherCAT)/=+-EP2338_05_00
//     PlcTask Inputs/GVL_SXR_VAC.fb_TV2K0_VGC_1.i_xClsLS <-> Channel 2/GVL_SXR_VAC.fb_TV2K0_VGC_1.i_xClsLS
//     PlcTask Inputs/GVL_SXR_VAC.fb_TV2K0_VGC_1.i_xOpnLS <-> Channel 1/GVL_SXR_VAC.fb_TV2K0_VGC_1.i_xOpnLS
//     PlcTask Outputs/GVL_SXR_VAC.fb_TV2K0_VGC_1.q_xOPN_DO <-> Channel 11/GVL_SXR_VAC.fb_TV2K0_VGC_1.q_xOPN_DO
//   plc_kfe_vac/plc_kfe_vac Instance <-> Device 1 (EtherCAT)/=+-EP2338_06_00
//     PlcTask Inputs/GVL_SXR_VAC.fb_MR1K1_BEND_VGC_1.i_xClsLS <-> Channel 2/GVL_SXR_VAC.fb_MR1K1_BEND_VGC_1.i_xClsLS
//     PlcTask Inputs/GVL_SXR_VAC.fb_MR1K1_BEND_VGC_1.i_xOpnLS <-> Channel 1/GVL_SXR_VAC.fb_MR1K1_BEND_VGC_1.i_xOpnLS
//     PlcTask Outputs/GVL_SXR_VAC.fb_MR1K1_BEND_VGC_1.q_xOPN_DO <-> Channel 11/GVL_SXR_VAC.fb_MR1K1_BEND_VGC_1.q_xOPN_DO
//   plc_kfe_vac/plc_kfe_vac Instance <-> Device 1 (EtherCAT)/=+-EP2338_07_00
//     PlcTask Inputs/GVL_SXR_VAC.fb_MR1K3_TXI_VGC_1.i_xClsLS <-> Channel 2/GVL_SXR_VAC.fb_MR1K3_TXI_VGC_1.i_xClsLS
//     PlcTask Inputs/GVL_SXR_VAC.fb_MR1K3_TXI_VGC_1.i_xOpnLS <-> Channel 1/GVL_SXR_VAC.fb_MR1K3_TXI_VGC_1.i_xOpnLS
//     PlcTask Outputs/GVL_SXR_VAC.fb_MR1K3_TXI_VGC_1.q_xOPN_DO <-> Channel 11/GVL_SXR_VAC.fb_MR1K3_TXI_VGC_1.q_xOPN_DO
//   plc_kfe_vac/plc_kfe_vac Instance <-> Device 1 (EtherCAT)/=+-EP2338_08_00
//     PlcTask Inputs/GVL_SXR_VAC.fb_SP1K1_MONO_VGC_1.i_xClsLS <-> Channel 2/GVL_SXR_VAC.fb_SP1K1_MONO_VGC_1.i_xClsLS
//     PlcTask Inputs/GVL_SXR_VAC.fb_SP1K1_MONO_VGC_1.i_xOpnLS <-> Channel 1/GVL_SXR_VAC.fb_SP1K1_MONO_VGC_1.i_xOpnLS
//     PlcTask Outputs/GVL_SXR_VAC.fb_SP1K1_MONO_VGC_1.q_xOPN_DO <-> Channel 11/GVL_SXR_VAC.fb_SP1K1_MONO_VGC_1.q_xOPN_DO
//   plc_kfe_vac/plc_kfe_vac Instance <-> Device 1 (EtherCAT)/=+-EP2338_09_02
//     PlcTask Inputs/GVL_SXR_VAC.fb_SP1K1_MONO_VGC_2.i_xClsLS <-> Channel 2/GVL_SXR_VAC.fb_SP1K1_MONO_VGC_2.i_xClsLS
//     PlcTask Inputs/GVL_SXR_VAC.fb_SP1K1_MONO_VGC_2.i_xOpnLS <-> Channel 1/GVL_SXR_VAC.fb_SP1K1_MONO_VGC_2.i_xOpnLS
//     PlcTask Outputs/GVL_SXR_VAC.fb_SP1K1_MONO_VGC_2.q_xOPN_DO <-> Channel 11/GVL_SXR_VAC.fb_SP1K1_MONO_VGC_2.q_xOPN_DO
//   plc_kfe_vac/plc_kfe_vac Instance <-> Device 1 (EtherCAT)/=+-EP2338_09_03
//     PlcTask Inputs/GVL_SXR_VAC.fb_IM1K3_PPM_VGC_1.i_xClsLS <-> Channel 2/GVL_SXR_VAC.fb_IM1K3_PPM_VGC_1.i_xClsLS
//     PlcTask Inputs/GVL_SXR_VAC.fb_IM1K3_PPM_VGC_1.i_xOpnLS <-> Channel 1/GVL_SXR_VAC.fb_IM1K3_PPM_VGC_1.i_xOpnLS
//     PlcTask Inputs/GVL_SXR_VAC.fb_TV3K0_VGC_1.i_xClsLS <-> Channel 6/GVL_SXR_VAC.fb_TV3K0_VGC_1.i_xClsLS
//     PlcTask Inputs/GVL_SXR_VAC.fb_TV3K0_VGC_1.i_xOpnLS <-> Channel 5/GVL_SXR_VAC.fb_TV3K0_VGC_1.i_xOpnLS
//     PlcTask Outputs/GVL_SXR_VAC.fb_IM1K3_PPM_VGC_1.q_xOPN_DO <-> Channel 11/GVL_SXR_VAC.fb_IM1K3_PPM_VGC_1.q_xOPN_DO
//     PlcTask Outputs/GVL_SXR_VAC.fb_TV3K0_VGC_1.q_xOPN_DO <-> Channel 15/GVL_SXR_VAC.fb_TV3K0_VGC_1.q_xOPN_DO
//   plc_kfe_vac/plc_kfe_vac Instance <-> Device 1 (EtherCAT)/=+-EP2338_10_02
//     PlcTask Inputs/GVL_SXR_VAC.fb_MR1K4_SOMS_VGC_1.i_xClsLS <-> Channel 2/GVL_SXR_VAC.fb_MR1K4_SOMS_VGC_1.i_xClsLS
//     PlcTask Inputs/GVL_SXR_VAC.fb_MR1K4_SOMS_VGC_1.i_xOpnLS <-> Channel 1/GVL_SXR_VAC.fb_MR1K4_SOMS_VGC_1.i_xOpnLS
//     PlcTask Outputs/GVL_SXR_VAC.fb_MR1K4_SOMS_VGC_1.q_xOPN_DO <-> Channel 11/GVL_SXR_VAC.fb_MR1K4_SOMS_VGC_1.q_xOPN_DO
//   plc_kfe_vac/plc_kfe_vac Instance <-> Device 1 (EtherCAT)/=+-EP2624_07_02
//     PlcTask Outputs/GVL_SXR_VAC.fb_MR1K1_BEND_GCC_1.q_xHV_DIS <-> Channel 2/GVL_SXR_VAC.fb_MR1K1_BEND_GCC_1.q_xHV_DIS
//     PlcTask Outputs/GVL_SXR_VAC.fb_MR1K3_TXI_GCC_1.q_xHV_DIS <-> Channel 1/GVL_SXR_VAC.fb_MR1K3_TXI_GCC_1.q_xHV_DIS
//   plc_kfe_vac/plc_kfe_vac Instance <-> Device 1 (EtherCAT)/=+-EP2624_08_02
//     PlcTask Outputs/GVL_SXR_VAC.fb_MR2K3_TXI_GCC_1.q_xHV_DIS <-> Channel 1/GVL_SXR_VAC.fb_MR2K3_TXI_GCC_1.q_xHV_DIS
//     PlcTask Outputs/GVL_SXR_VAC.fb_SP1K1_MONO_GCC_1.q_xHV_DIS <-> Channel 2/GVL_SXR_VAC.fb_SP1K1_MONO_GCC_1.q_xHV_DIS
//   plc_kfe_vac/plc_kfe_vac Instance <-> Device 1 (EtherCAT)/=+-EP2624_10_01
//     PlcTask Outputs/GVL_SXR_VAC.fb_MR1K4_SOMS_GCC_1.q_xHV_DIS <-> Channel 2/GVL_SXR_VAC.fb_MR1K4_SOMS_GCC_1.q_xHV_DIS
//     PlcTask Outputs/GVL_SXR_VAC.fb_TV3K0_GCC_1.q_xHV_DIS <-> Channel 1/GVL_SXR_VAC.fb_TV3K0_GCC_1.q_xHV_DIS
//   plc_kfe_vac/plc_kfe_vac Instance <-> Device 1 (EtherCAT)/=+-EP3174_07_01
//     PlcTask Inputs/GVL_SXR_VAC.fb_MR1K1_BEND_GCC_1.i_iPRESS_R <-> AI Standard Channel 4/GVL_SXR_VAC.fb_MR1K1_BEND_GCC_1.i_iPRESS_R
//     PlcTask Inputs/GVL_SXR_VAC.fb_MR1K1_BEND_GPI_1.i_iPRESS_R <-> AI Standard Channel 3/GVL_SXR_VAC.fb_MR1K1_BEND_GPI_1.i_iPRESS_R
//     PlcTask Inputs/GVL_SXR_VAC.fb_MR1K3_TXI_GCC_1.i_iPRESS_R <-> AI Standard Channel 2/GVL_SXR_VAC.fb_MR1K3_TXI_GCC_1.i_iPRESS_R
//     PlcTask Inputs/GVL_SXR_VAC.fb_MR1K3_TXI_GPI_1.i_iPRESS_R <-> AI Standard Channel 1/GVL_SXR_VAC.fb_MR1K3_TXI_GPI_1.i_iPRESS_R
//   plc_kfe_vac/plc_kfe_vac Instance <-> Device 1 (EtherCAT)/=+-EP3174_08_01
//     PlcTask Inputs/GVL_SXR_VAC.fb_MR2K3_TXI_GCC_1.i_iPRESS_R <-> AI Standard Channel 2/GVL_SXR_VAC.fb_MR2K3_TXI_GCC_1.i_iPRESS_R
//     PlcTask Inputs/GVL_SXR_VAC.fb_MR2K3_TXI_GPI_1.i_iPRESS_R <-> AI Standard Channel 1/GVL_SXR_VAC.fb_MR2K3_TXI_GPI_1.i_iPRESS_R
//     PlcTask Inputs/GVL_SXR_VAC.fb_SP1K1_MONO_GCC_1.i_iPRESS_R <-> AI Standard Channel 4/GVL_SXR_VAC.fb_SP1K1_MONO_GCC_1.i_iPRESS_R
//     PlcTask Inputs/GVL_SXR_VAC.fb_SP1K1_MONO_GPI_1.i_iPRESS_R <-> AI Standard Channel 3/GVL_SXR_VAC.fb_SP1K1_MONO_GPI_1.i_iPRESS_R
//   plc_kfe_vac/plc_kfe_vac Instance <-> Device 1 (EtherCAT)/=+-EP3174_10_00
//     PlcTask Inputs/GVL_SXR_VAC.fb_MR1K4_SOMS_GCC_1.i_iPRESS_R <-> AI Standard Channel 3/Value
//     PlcTask Inputs/GVL_SXR_VAC.fb_MR1K4_SOMS_GPI_1.i_iPRESS_R <-> AI Standard Channel 2/GVL_SXR_VAC.fb_MR1K4_SOMS_GPI_1.i_iPRESS_R
//     PlcTask Inputs/GVL_SXR_VAC.fb_TV3K0_GCC_1.i_iPRESS_R <-> AI Standard Channel 1/GVL_SXR_VAC.fb_TV3K0_GCC_1.i_iPRESS_R
//     PlcTask Inputs/GVL_SXR_VAC.fb_TV3K0_GPI_1.i_iPRESS_R <-> AI Standard Channel 4/GVL_SXR_VAC.fb_TV3K0_GPI_1.i_iPRESS_R
//   plc_kfe_vac/plc_kfe_vac Instance <-> SimDevice 2 (EtherCAT Simulation)/=+-ES2004_03_03
//     PlcTask Outputs/GVL_SXR_VAC.fb_IM1K0_XTES_VGC_1.q_xOPN_DO <-> Channel 3/Output
//     PlcTask Outputs/GVL_SXR_VAC.fb_IM1K0_XTES_VGC_1.q_xOPN_DO <-> Channel 4/Output
//   plc_kfe_vac/plc_kfe_vac Instance <-> plc_kfe_vac/plc_kfe_vac Instance
//     FSV_task Outputs/GVL_VFS.fb_TV2K0_VFS_1.q_xMPS_OK <-> PlcTask Inputs/GVL_SXR_VAC.fb_TV2K0_VFS_1_Interface.i_xMPS_OK
//     PlcTask Inputs/GVL_SXR_VAC.fb_TV2K0_VFS_1_Interface.i_eVFS_State <-> FSV_task Outputs/GVL_VFS.fb_TV2K0_VFS_1.q_eVFS_State
//     PlcTask Inputs/GVL_SXR_VAC.fb_TV2K0_VFS_1_Interface.i_xTrigger <-> FSV_task Outputs/GVL_VFS.fb_TV2K0_VFS_1.q_xTrigger
//     PlcTask Inputs/GVL_SXR_VAC.fb_TV2K0_VFS_1_Interface.i_xVAC_FAULT_OK <-> FSV_task Outputs/GVL_VFS.fb_TV2K0_VFS_1.q_xVAC_FAULT_OK
//     PlcTask Inputs/GVL_SXR_VAC.fb_TV2K0_VFS_1_Interface.i_xVFS_Closed <-> FSV_task Outputs/GVL_VFS.fb_TV2K0_VFS_1.q_xVFS_Closed
//     PlcTask Inputs/GVL_SXR_VAC.fb_TV2K0_VFS_1_Interface.i_xVFS_Open <-> FSV_task Outputs/GVL_VFS.fb_TV2K0_VFS_1.q_xVFS_Open
//     PlcTask Outputs/GVL_SXR_VAC.fb_TV2K0_VFS_1_Interface.q_xCLS_SW <-> FSV_task Inputs/GVL_VFS.fb_TV2K0_VFS_1.i_xCLS_SW
//     PlcTask Outputs/GVL_SXR_VAC.fb_TV2K0_VFS_1_Interface.q_xOPN_SW <-> FSV_task Inputs/GVL_VFS.fb_TV2K0_VFS_1.i_xOPN_SW
//     PlcTask Outputs/GVL_SXR_VAC.fb_TV2K0_VFS_1_Interface.q_xOverrideMode <-> FSV_task Inputs/GVL_VFS.fb_TV2K0_VFS_1.i_xOverrideMode
//     PlcTask Outputs/GVL_SXR_VAC.fb_TV2K0_VFS_1_Interface.q_xOverrideOpen <-> FSV_task Inputs/GVL_VFS.fb_TV2K0_VFS_1.i_xOverrideOpen
//     PlcTask Outputs/GVL_SXR_VAC.fb_TV2K0_VFS_1_Interface.q_xPRESS_OK <-> FSV_task Inputs/GVL_VFS.fb_TV2K0_VFS_1.i_xPress_OK
//     PlcTask Outputs/GVL_SXR_VAC.fb_TV2K0_VFS_1_Interface.q_xVAC_FAULT_Reset <-> FSV_task Inputs/GVL_VFS.fb_TV2K0_VFS_1.i_xVAC_FAULT_Reset
//   plc_kfe_vac_sim/plc_kfe_vac_sim Instance <-> SimDevice 2 (EtherCAT Simulation)/=+-EL2794_00_03
//     SimTask Inputs/GVL_SXR_VAC.st_RTDSK0_PIP_{1..4}.xOn <-> Channel {1..4}/GVL_SXR_VAC.fb_RTDSK0_PIP_{1..4}.q_xHVEna_DO  (4 links)
//   plc_kfe_vac_sim/plc_kfe_vac_sim Instance <-> SimDevice 2 (EtherCAT Simulation)/=+-EL2794_00_06
//     SimTask Inputs/GVL_SXR_VAC.st_PCPM3B_PIP_1.xOn <-> Channel 2/GVL_SXR_VAC.fb_PCPM3B_PIP_1.q_xHVEna_DO
//     SimTask Inputs/GVL_SXR_VAC.st_RTDSK0_PIP_5.xOn <-> Channel 1/GVL_SXR_VAC.fb_RTDSK0_PIP_5.q_xHVEna_DO
//   plc_kfe_vac_sim/plc_kfe_vac_sim Instance <-> SimDevice 2 (EtherCAT Simulation)/=+-EL2794_00_10
//     SimTask Inputs/GVL_SXR_VAC.st_MR1K1_BEND_PIP_1.xOn <-> Channel 3/GVL_SXR_VAC.fb_MR1K1_BEND_PIP_1.q_xHVEna_DO
//     SimTask Inputs/GVL_SXR_VAC.st_MR1K3_TXI_PIP_1.xOn <-> Channel 4/GVL_SXR_VAC.fb_MR1K3_TXI_PIP_1.q_xHVEna_DO
//     SimTask Inputs/GVL_SXR_VAC.st_PA1K0_PIP_1.xOn <-> Channel 1/GVL_SXR_VAC.fb_PA1K0_PIP_1.q_xHVEna_DO
//   plc_kfe_vac_sim/plc_kfe_vac_sim Instance <-> SimDevice 2 (EtherCAT Simulation)/=+-EL2794_00_13
//     SimTask Inputs/GVL_SXR_VAC.st_MR2K3_TXI_PIP_1.xOn <-> Channel 1/GVL_SXR_VAC.fb_MR2K3_TXI_PIP_1.q_xHVEna_DO
//     SimTask Inputs/GVL_SXR_VAC.st_SP1K1_MONO_PIP_1.xOn <-> Channel 2/GVL_SXR_VAC.fb_SP1K1_MONO_PIP_1.q_xHVEna_DO
//     SimTask Inputs/GVL_SXR_VAC.st_SP1K1_MONO_PIP_2.xOn <-> Channel 3/GVL_SXR_VAC.fb_SP1K1_MONO_PIP_2.q_xHVEna_DO
//     SimTask Inputs/GVL_SXR_VAC.st_TV3K0_PIP_1.xOn <-> Channel 4/GVL_SXR_VAC.fb_TV3K0_PIP_1.q_xHVEna_DO
//   plc_kfe_vac_sim/plc_kfe_vac_sim Instance <-> SimDevice 2 (EtherCAT Simulation)/=+-EL2794_15_03
//     SimTask Inputs/GVL_SXR_VAC.st_MR1K4_SOMS_PIP_1.xOn <-> Channel 1/GVL_SXR_VAC.fb_MR1K4_SOMS_PIP_1.q_xHVEna_DO
//     SimTask Inputs/GVL_SXR_VAC.st_ST1K4_TEST_PIP_1.xOn <-> Channel 2/GVL_SXR_VAC.fb_ST1K4_TEST_PIP_1.q_xHVEna_DO
//     SimTask Inputs/GVL_SXR_VAC.st_ST2K4_BCS_PIP_1.xOn <-> Channel 3/GVL_SXR_VAC.fb_ST2K4_BCS_PIP_1.q_xHVEna_DO
//     SimTask Inputs/GVL_SXR_VAC.st_ST3K4_PPS_PIP_1.xOn <-> Channel 4/GVL_SXR_VAC.fb_ST3K4_PPS_PIP_1.q_xHVEna_DO
//   plc_kfe_vac_sim/plc_kfe_vac_sim Instance <-> SimDevice 2 (EtherCAT Simulation)/=+-EL2794_15_06
//     SimTask Inputs/GVL_SXR_VAC.st_PC4K4_XTES_PIP_1.xOn <-> Channel 1/GVL_SXR_VAC.fb_PC4K4_XTES_PIP_1.q_xHVEna_DO
//   plc_kfe_vac_sim/plc_kfe_vac_sim Instance <-> SimDevice 2 (EtherCAT Simulation)/=+-EL2798_01_02
//     SimTask Inputs/GVL_SXR_VAC.st_DMPS_GCC_1.i_xHvOn <-> Channel 1/GVL_SXR_VAC.fb_DMPS_GCC_1.q_xHV_DIS
//     SimTask Inputs/GVL_SXR_VAC.st_IM2K0_XTES_GCC_1.i_xHvOn <-> Channel 2/GVL_SXR_VAC.fb_IM2K0_XTES_GCC_1.q_xHV_DIS
//     SimTask Inputs/GVL_SXR_VAC.st_PCPM3B_GFS_1.i_xHvOn <-> Channel 5/GVL_SXR_VAC.fb_PCPM3B_GFS_1.q_xHV_DIS
//     SimTask Inputs/GVL_SXR_VAC.st_SL1K0_GCC_1.i_xHvOn <-> Channel 4/GVL_SXR_VAC.fb_SL1K0_GCC_1.q_xHV_DIS
//   plc_kfe_vac_sim/plc_kfe_vac_sim Instance <-> SimDevice 2 (EtherCAT Simulation)/=+-EL2798_01_06
//     SimTask Inputs/GVL_SXR_VAC.st_MR1K1_BEND_GCC_1.i_xHvOn <-> Channel 5/GVL_SXR_VAC.fb_MR1K1_BEND_GCC_1.q_xHV_DIS
//     SimTask Inputs/GVL_SXR_VAC.st_PA1K0_GCC_1.i_xHvOn <-> Channel 4/GVL_SXR_VAC.fb_PA1K0_GCC_1.q_xHV_DIS
//     SimTask Inputs/GVL_SXR_VAC.st_TV2K0_GCC_1.i_xHvOn <-> Channel 1/GVL_SXR_VAC.fb_TV2K0_GCC_1.q_xHV_DIS
//     SimTask Inputs/GVL_SXR_VAC.st_TV2K0_GCC_2.i_xHvOn <-> Channel 2/GVL_SXR_VAC.fb_TV2K0_GCC_2.q_xHV_DIS
//   plc_kfe_vac_sim/plc_kfe_vac_sim Instance <-> SimDevice 2 (EtherCAT Simulation)/=+-EP2338_04_00
//     SimTask Inputs/GVL_SXR_VAC.st_EM1K0_XGMD_VGC_1.i_xSol <-> Channel 11/GVL_SXR_VAC.fb_EM1K0_XGMD_VGC_1.q_xOPN_DO
//     SimTask Inputs/GVL_SXR_VAC.st_EM1K0_XGMD_VGC_2.i_xSol <-> Channel 15/GVL_SXR_VAC.fb_EM1K0_XGMD_VGC_2.q_xOPN_DO
//     SimTask Outputs/GVL_SXR_VAC.st_EM1K0_XGMD_VGC_1.q_xClsLS <-> Channel 2/GVL_SXR_VAC.fb_EM1K0_XGMD_VGC_1.i_xClsLS
//     SimTask Outputs/GVL_SXR_VAC.st_EM1K0_XGMD_VGC_2.q_xClsLS <-> Channel 6/GVL_SXR_VAC.fb_EM1K0_XGMD_VGC_2.i_xClsLS
//     SimTask Outputs/GVL_SXR_VAC.st_EM1K0_XGMD_VGC_1.q_xOpnLS <-> Channel 1/GVL_SXR_VAC.fb_EM1K0_XGMD_VGC_1.i_xOpnLS
//     SimTask Outputs/GVL_SXR_VAC.st_EM1K0_XGMD_VGC_2.q_xOpnLS <-> Channel 5/GVL_SXR_VAC.fb_EM1K0_XGMD_VGC_2.i_xOpnLS
//   plc_kfe_vac_sim/plc_kfe_vac_sim Instance <-> SimDevice 2 (EtherCAT Simulation)/=+-EP2338_05_00
//     SimTask Inputs/GVL_SXR_VAC.st_TV2K0_VGC_1.i_xSol <-> Channel 11/GVL_SXR_VAC.fb_TV2K0_VGC_1.q_xOPN_DO
//     SimTask Outputs/GVL_SXR_VAC.st_TV2K0_VGC_1.q_xClsLS <-> Channel 2/GVL_SXR_VAC.fb_TV2K0_VGC_1.i_xClsLS
//     SimTask Outputs/GVL_SXR_VAC.st_TV2K0_VGC_1.q_xOpnLS <-> Channel 1/GVL_SXR_VAC.fb_TV2K0_VGC_1.i_xOpnLS
//   plc_kfe_vac_sim/plc_kfe_vac_sim Instance <-> SimDevice 2 (EtherCAT Simulation)/=+-EP2338_06_00
//     SimTask Inputs/GVL_SXR_VAC.st_MR1K1_BEND_VGC_1.i_xSol <-> Channel 11/GVL_SXR_VAC.fb_MR1K1_BEND_VGC_1.q_xOPN_DO
//     SimTask Outputs/GVL_SXR_VAC.st_MR1K1_BEND_VGC_1.q_xClsLS <-> Channel 2/GVL_SXR_VAC.fb_MR1K1_BEND_VGC_1.i_xClsLS
//     SimTask Outputs/GVL_SXR_VAC.st_MR1K1_BEND_VGC_1.q_xOpnLS <-> Channel 1/GVL_SXR_VAC.fb_MR1K1_BEND_VGC_1.i_xOpnLS
//   plc_kfe_vac_sim/plc_kfe_vac_sim Instance <-> SimDevice 2 (EtherCAT Simulation)/=+-EP2338_07_00
//     SimTask Inputs/GVL_SXR_VAC.st_MR1K3_TXI_VGC_1.i_xSol <-> Channel 11/GVL_SXR_VAC.fb_MR1K3_TXI_VGC_1.q_xOPN_DO
//     SimTask Outputs/GVL_SXR_VAC.st_MR1K3_TXI_VGC_1.q_xClsLS <-> Channel 2/GVL_SXR_VAC.fb_MR1K3_TXI_VGC_1.i_xClsLS
//     SimTask Outputs/GVL_SXR_VAC.st_MR1K3_TXI_VGC_1.q_xOpnLS <-> Channel 1/GVL_SXR_VAC.fb_MR1K3_TXI_VGC_1.i_xOpnLS
//   plc_kfe_vac_sim/plc_kfe_vac_sim Instance <-> SimDevice 2 (EtherCAT Simulation)/=+-EP2338_08_00
//     SimTask Inputs/GVL_SXR_VAC.st_SP1K1_MONO_VGC_1.i_xSol <-> Channel 11/GVL_SXR_VAC.fb_SP1K1_MONO_VGC_1.q_xOPN_DO
//     SimTask Outputs/GVL_SXR_VAC.st_SP1K1_MONO_VGC_1.q_xClsLS <-> Channel 2/GVL_SXR_VAC.fb_SP1K1_MONO_VGC_1.i_xClsLS
//     SimTask Outputs/GVL_SXR_VAC.st_SP1K1_MONO_VGC_1.q_xOpnLS <-> Channel 1/GVL_SXR_VAC.fb_SP1K1_MONO_VGC_1.i_xOpnLS
//   plc_kfe_vac_sim/plc_kfe_vac_sim Instance <-> SimDevice 2 (EtherCAT Simulation)/=+-EP2338_09_02
//     SimTask Inputs/GVL_SXR_VAC.st_SP1K1_MONO_VGC_2.i_xSol <-> Channel 11/GVL_SXR_VAC.fb_SP1K1_MONO_VGC_2.q_xOPN_DO
//     SimTask Outputs/GVL_SXR_VAC.st_SP1K1_MONO_VGC_2.q_xClsLS <-> Channel 2/GVL_SXR_VAC.fb_SP1K1_MONO_VGC_2.i_xClsLS
//     SimTask Outputs/GVL_SXR_VAC.st_SP1K1_MONO_VGC_2.q_xOpnLS <-> Channel 1/GVL_SXR_VAC.fb_SP1K1_MONO_VGC_2.i_xOpnLS
//   plc_kfe_vac_sim/plc_kfe_vac_sim Instance <-> SimDevice 2 (EtherCAT Simulation)/=+-EP2338_09_03
//     SimTask Inputs/GVL_SXR_VAC.st_IM1K2_PPM_VGC_1.i_xSol <-> Channel 11/GVL_SXR_VAC.fb_IM1K2_PPM_VGC_1.q_xOPN_DO
//     SimTask Inputs/GVL_SXR_VAC.st_TV3K0_VGC_1.i_xSol <-> Channel 15/GVL_SXR_VAC.fb_TV3K0_VGC_1.q_xOPN_DO
//     SimTask Outputs/GVL_SXR_VAC.st_IM1K2_PPM_VGC_1.q_xClsLS <-> Channel 2/GVL_SXR_VAC.fb_IM1K2_PPM_VGC_1.i_xClsLS
//     SimTask Outputs/GVL_SXR_VAC.st_IM1K2_PPM_VGC_1.q_xOpnLS <-> Channel 1/GVL_SXR_VAC.fb_IM1K2_PPM_VGC_1.i_xOpnLS
//     SimTask Outputs/GVL_SXR_VAC.st_TV3K0_VGC_1.q_xClsLS <-> Channel 6/GVL_SXR_VAC.fb_TV3K0_VGC_1.i_xClsLS
//     SimTask Outputs/GVL_SXR_VAC.st_TV3K0_VGC_1.q_xOpnLS <-> Channel 5/GVL_SXR_VAC.fb_TV3K0_VGC_1.i_xOpnLS
//   plc_kfe_vac_sim/plc_kfe_vac_sim Instance <-> SimDevice 2 (EtherCAT Simulation)/=+-EP2338_10_02
//     SimTask Inputs/GVL_SXR_VAC.st_MR1K4_SOMS_VGC_1.i_xSol <-> Channel 11/GVL_SXR_VAC.fb_MR1K4_SOMS_VGC_1.q_xOPN_DO
//     SimTask Outputs/GVL_SXR_VAC.st_MR1K4_SOMS_VGC_1.q_xClsLS <-> Channel 2/GVL_SXR_VAC.fb_MR1K4_SOMS_VGC_1.i_xClsLS
//     SimTask Outputs/GVL_SXR_VAC.st_MR1K4_SOMS_VGC_1.q_xOpnLS <-> Channel 1/GVL_SXR_VAC.fb_MR1K4_SOMS_VGC_1.i_xOpnLS
//   plc_kfe_vac_sim/plc_kfe_vac_sim Instance <-> SimDevice 2 (EtherCAT Simulation)/=+-EP2338_11_02
//     SimTask Inputs/GVL_SXR_VAC.st_TV1K4_VGC_1.i_xSol <-> Channel 11/GVL_SXR_VAC.fb_TV1K4_VGC_1.q_xOPN_DO
//     SimTask Inputs/GVL_SXR_VAC.st_TV1K4_VGC_2.i_xSol <-> Channel 15/GVL_SXR_VAC.fb_TV1K4_VGC_2.q_xOPN_DO
//     SimTask Outputs/GVL_SXR_VAC.st_TV1K4_VGC_1.q_xClsLS <-> Channel 2/GVL_SXR_VAC.fb_TV1K4_VGC_1.i_xClsLS
//     SimTask Outputs/GVL_SXR_VAC.st_TV1K4_VGC_2.q_xClsLS <-> Channel 6/GVL_SXR_VAC.fb_TV1K4_VGC_2.i_xClsLS
//     SimTask Outputs/GVL_SXR_VAC.st_TV1K4_VGC_1.q_xOpnLS <-> Channel 1/GVL_SXR_VAC.fb_TV1K4_VGC_1.i_xOpnLS
//     SimTask Outputs/GVL_SXR_VAC.st_TV1K4_VGC_2.q_xOpnLS <-> Channel 5/GVL_SXR_VAC.fb_TV1K4_VGC_2.i_xOpnLS
//   plc_kfe_vac_sim/plc_kfe_vac_sim Instance <-> SimDevice 2 (EtherCAT Simulation)/=+-EP2338_14_00
//     SimTask Inputs/GVL_SXR_VAC.st_ST3K4_XTES_VGC_1.i_xSol <-> Channel 11/GVL_SXR_VAC.fb_ST3K4_XTES_VGC_1.q_xOPN_DO
//     SimTask Outputs/GVL_SXR_VAC.st_ST3K4_XTES_VGC_1.q_xClsLS <-> Channel 2/GVL_SXR_VAC.fb_ST3K4_XTES_VGC_1.i_xClsLS
//     SimTask Outputs/GVL_SXR_VAC.st_ST3K4_XTES_VGC_1.q_xOpnLS <-> Channel 1/GVL_SXR_VAC.fb_ST3K4_XTES_VGC_1.i_xOpnLS
//   plc_kfe_vac_sim/plc_kfe_vac_sim Instance <-> SimDevice 2 (EtherCAT Simulation)/=+-EP2624_07_02
//     SimTask Inputs/GVL_SXR_VAC.st_MR1K3_TXI_GCC_1.i_xHvOn <-> Channel 1/GVL_SXR_VAC.fb_MR1K3_TXI_GCC_1.q_xHV_DIS
//   plc_kfe_vac_sim/plc_kfe_vac_sim Instance <-> SimDevice 2 (EtherCAT Simulation)/=+-EP2624_08_02
//     SimTask Inputs/GVL_SXR_VAC.st_MR2K3_TXI_GCC_1.i_xHvOn <-> Channel 1/GVL_SXR_VAC.fb_MR2K3_TXI_GCC_1.q_xHV_DIS
//   plc_kfe_vac_sim/plc_kfe_vac_sim Instance <-> SimDevice 2 (EtherCAT Simulation)/=+-EP2624_09_01
//     SimTask Inputs/GVL_SXR_VAC.st_SP1K1_MONO_GCC_1.i_xHvOn <-> Channel 1/GVL_SXR_VAC.fb_SP1K1_MONO_GCC_1.q_xHV_DIS
//   plc_kfe_vac_sim/plc_kfe_vac_sim Instance <-> SimDevice 2 (EtherCAT Simulation)/=+-EP2624_10_01
//     SimTask Inputs/GVL_SXR_VAC.st_TV3K0_GCC_1.i_xHvOn <-> Channel 1/GVL_SXR_VAC.fb_TV3K0_GCC_1.q_xHV_DIS
//   plc_kfe_vac_sim/plc_kfe_vac_sim Instance <-> SimDevice 2 (EtherCAT Simulation)/=+-EP2624_11_01
//     SimTask Inputs/GVL_SXR_VAC.st_MR1K4_SOMS_GCC_1.i_xHvOn <-> Channel 2/GVL_SXR_VAC.fb_MR1K4_SOMS_GCC_1.q_xHV_DIS
//     SimTask Inputs/GVL_SXR_VAC.st_TV1K4_GCC_1.i_xHvOn <-> Channel 1/GVL_SXR_VAC.fb_TV1K4_GCC_1.q_xHV_DIS
//   plc_kfe_vac_sim/plc_kfe_vac_sim Instance <-> SimDevice 2 (EtherCAT Simulation)/=+-EP2624_12_01
//     SimTask Inputs/GVL_SXR_VAC.st_ST1K4_TEST_GCC_1.i_xHvOn <-> Channel 1/GVL_SXR_VAC.fb_ST1K4_TEST_GCC_1.q_xHV_DIS
//   plc_kfe_vac_sim/plc_kfe_vac_sim Instance <-> SimDevice 2 (EtherCAT Simulation)/=+-EP2624_13_01
//     SimTask Inputs/GVL_SXR_VAC.st_ST2K4_BCS_GCC_1.i_xHvOn <-> Channel 1/GVL_SXR_VAC.fb_ST2K4_BCS_GCC_1.q_xHV_DIS
//   plc_kfe_vac_sim/plc_kfe_vac_sim Instance <-> SimDevice 2 (EtherCAT Simulation)/=+-EP2624_14_02
//     SimTask Inputs/GVL_SXR_VAC.st_PC4K4_XTES_GCC_1.i_xHvOn <-> Channel 1/GVL_SXR_VAC.fb_PC4K4_XTES_GCC_1.q_xHV_DIS
//   plc_kfe_vac_sim/plc_kfe_vac_sim Instance <-> SimDevice 2 (EtherCAT Simulation)/=+-EP3174_07_01
//     SimTask Outputs/GVL_SXR_VAC.st_MR1K3_TXI_GCC_1.q_iRawPress <-> AI Standard Channel 2/GVL_SXR_VAC.fb_MR1K3_TXI_GCC_1.i_iPRESS_R
//     SimTask Outputs/GVL_SXR_VAC.st_MR1K3_TXI_GPI_1.q_iRawPress <-> AI Standard Channel 1/GVL_SXR_VAC.fb_MR1K3_TXI_GPI_1.i_iPRESS_R
//   plc_kfe_vac_sim/plc_kfe_vac_sim Instance <-> SimDevice 2 (EtherCAT Simulation)/=+-EP3174_08_01
//     SimTask Outputs/GVL_SXR_VAC.st_MR2K3_TXI_GCC_1.q_iRawPress <-> AI Standard Channel 2/GVL_SXR_VAC.fb_MR2K3_TXI_GCC_1.i_iPRESS_R
//     SimTask Outputs/GVL_SXR_VAC.st_MR2K3_TXI_GPI_1.q_iRawPress <-> AI Standard Channel 1/GVL_SXR_VAC.fb_MR2K3_TXI_GPI_1.i_iPRESS_R
//   plc_kfe_vac_sim/plc_kfe_vac_sim Instance <-> SimDevice 2 (EtherCAT Simulation)/=+-EP3174_09_00
//     SimTask Outputs/GVL_SXR_VAC.st_SP1K1_MONO_GCC_1.q_iRawPress <-> AI Standard Channel 1/GVL_SXR_VAC.fb_SP1K1_MONO_GCC_1.i_iPRESS_R
//     SimTask Outputs/GVL_SXR_VAC.st_SP1K1_MONO_GPI_1.q_iRawPress <-> AI Standard Channel 2/GVL_SXR_VAC.fb_SP1K1_MONO_GPI_1.i_iPRESS_R
//   plc_kfe_vac_sim/plc_kfe_vac_sim Instance <-> SimDevice 2 (EtherCAT Simulation)/=+-EP3174_10_00
//     SimTask Outputs/GVL_SXR_VAC.st_MR1K4_SOMS_GPI_1.q_iRawPress <-> AI Standard Channel 2/GVL_SXR_VAC.fb_MR1K4_SOMS_GPI_1.i_iPRESS_R
//     SimTask Outputs/GVL_SXR_VAC.st_TV3K0_GCC_1.q_iRawPress <-> AI Standard Channel 1/GVL_SXR_VAC.fb_TV3K0_GCC_1.i_iPRESS_R
//     SimTask Outputs/GVL_SXR_VAC.st_TV3K0_GPI_1.q_iRawPress <-> AI Standard Channel 4/GVL_SXR_VAC.fb_TV3K0_GPI_1.i_iPRESS_R
//   plc_kfe_vac_sim/plc_kfe_vac_sim Instance <-> SimDevice 2 (EtherCAT Simulation)/=+-EP3174_11_00
//     SimTask Outputs/GVL_SXR_VAC.st_MR1K4_SOMS_GCC_1.q_iRawPress <-> AI Standard Channel 3/GVL_SXR_VAC.fb_MR1K4_SOMS_GCC_1.i_iPRESS_R
//     SimTask Outputs/GVL_SXR_VAC.st_TV1K4_GCC_1.q_iRawPress <-> AI Standard Channel 2/GVL_SXR_VAC.fb_TV1K4_GCC_1.i_iPRESS_R
//     SimTask Outputs/GVL_SXR_VAC.st_TV1K4_GPI_1.q_iRawPress <-> AI Standard Channel 1/GVL_SXR_VAC.fb_TV1K4_GPI_1.i_iPRESS_R
//   plc_kfe_vac_sim/plc_kfe_vac_sim Instance <-> SimDevice 2 (EtherCAT Simulation)/=+-EP3174_12_00
//     SimTask Outputs/GVL_SXR_VAC.st_ST1K4_TEST_GCC_1.q_iRawPress <-> AI Standard Channel 2/GVL_SXR_VAC.fb_ST1K4_TEST_GCC_1.i_iPRESS_R
//     SimTask Outputs/GVL_SXR_VAC.st_ST1K4_TEST_GPI_1.q_iRawPress <-> AI Standard Channel 1/GVL_SXR_VAC.fb_ST1K4_TEST_GPI_1.i_iPRESS_R
//   plc_kfe_vac_sim/plc_kfe_vac_sim Instance <-> SimDevice 2 (EtherCAT Simulation)/=+-EP3174_13_00
//     SimTask Outputs/GVL_SXR_VAC.st_ST2K4_BCS_GCC_1.q_iRawPress <-> AI Standard Channel 2/GVL_SXR_VAC.fb_ST2K4_BCS_GCC_1.i_iPRESS_R
//     SimTask Outputs/GVL_SXR_VAC.st_ST2K4_BCS_GPI_1.q_iRawPress <-> AI Standard Channel 1/GVL_SXR_VAC.fb_ST2K4_BCS_GPI_1.i_iPRESS_R
//   plc_kfe_vac_sim/plc_kfe_vac_sim Instance <-> SimDevice 2 (EtherCAT Simulation)/=+-EP3174_14_01
//     SimTask Outputs/GVL_SXR_VAC.st_PC4K4_XTES_GCC_1.q_iRawPress <-> AI Standard Channel 2/GVL_SXR_VAC.fb_PC4K4_XTES_GCC_1.i_iPRESS_R
//     SimTask Outputs/GVL_SXR_VAC.st_PC4K4_XTES_GPI_1.q_iRawPress <-> AI Standard Channel 1/GVL_SXR_VAC.fb_PC4K4_XTES_GPI_1.i_iPRESS_R
//   plc_kfe_vac_sim/plc_kfe_vac_sim Instance <-> SimDevice 2 (EtherCAT Simulation)/=+-ES1004_03_01
//     SimTask Outputs/GVL_SXR_VAC.st_EM1K0_GMD_VGC_1.q_xClsLS <-> Channel 4/GVL_SXR_VAC.fb_EM1K0_GMD_VGC_1.i_xClsLS
//     SimTask Outputs/GVL_SXR_VAC.st_EM1K0_GMD_VGC_1.q_xOpnLS <-> Channel 3/GVL_SXR_VAC.fb_EM1K0_GMD_VGC_1.i_xOpnLS
//     SimTask Outputs/GVL_SXR_VAC.st_RTDSK0_VGC_1.q_xClsLS <-> Channel 2/GVL_SXR_VAC.fb_RTDSK0_VGC_1.i_xClsLS
//     SimTask Outputs/GVL_SXR_VAC.st_RTDSK0_VGC_1.q_xOpnLS <-> Channel 1/GVL_SXR_VAC.fb_RTDSK0_VGC_1.i_xOpnLS
//   plc_kfe_vac_sim/plc_kfe_vac_sim Instance <-> SimDevice 2 (EtherCAT Simulation)/=+-ES1004_03_04
//     SimTask Outputs/GVL_SXR_VAC.st_AT1K0_GAS_VGC_1.q_xClsLS <-> Channel 2/GVL_SXR_VAC.fb_AT1K0_GAS_VGC_1.i_xClsLS
//     SimTask Outputs/GVL_SXR_VAC.st_AT1K0_GAS_VGC_1.q_xOpnLS <-> Channel 1/GVL_SXR_VAC.fb_AT1K0_GAS_VGC_1.i_xOpnLS
//   plc_kfe_vac_sim/plc_kfe_vac_sim Instance <-> SimDevice 2 (EtherCAT Simulation)/=+-ES2004_03_02
//     SimTask Inputs/GVL_SXR_VAC.st_EM1K0_GMD_VGC_1.i_xSol <-> Channel 3/GVL_SXR_VAC.fb_EM1K0_GMD_VGC_1.q_xOPN_DO
//     SimTask Inputs/GVL_SXR_VAC.st_RTDSK0_VGC_1.i_xSol <-> Channel 1/GVL_SXR_VAC.fb_RTDSK0_VGC_1.q_xOPN_DO
//   plc_kfe_vac_sim/plc_kfe_vac_sim Instance <-> SimDevice 2 (EtherCAT Simulation)/=+-ES2004_03_03
//     SimTask Inputs/GVL_SXR_VAC.st_AT1K0_GAS_VGC_1.i_xSol <-> Channel 1/GVL_SXR_VAC.fb_AT1K0_GAS_VGC_1.q_xOPN_DO
//   plc_kfe_vac_sim/plc_kfe_vac_sim Instance <-> SimDevice 2 (EtherCAT Simulation)/=+-ES3068_01_01
//     SimTask Outputs/GVL_SXR_VAC.st_DMPS_GCC_1.q_iRawPress <-> AI Standard Channel 1/GVL_SXR_VAC.fb_DMPS_GCC_1.i_iPRESS_R
//     SimTask Outputs/GVL_SXR_VAC.st_DMPS_GPI_1.q_iRawPress <-> AI Standard Channel 5/GVL_SXR_VAC.fb_DMPS_GPI_1.i_iPRESS_R
//     SimTask Outputs/GVL_SXR_VAC.st_IM2K0_XTES_GCC_1.q_iRawPress <-> AI Standard Channel 3/GVL_SXR_VAC.fb_IM2K0_XTES_GCC_1.i_iPRESS_R
//     SimTask Outputs/GVL_SXR_VAC.st_IM2K0_XTES_GPI_1.q_iRawPress <-> AI Standard Channel 6/GVL_SXR_VAC.fb_IM2K0_XTES_GPI_1.i_iPRESS_R
//   plc_kfe_vac_sim/plc_kfe_vac_sim Instance <-> SimDevice 2 (EtherCAT Simulation)/=+-ES3068_01_04
//     SimTask Outputs/GVL_SXR_VAC.st_PCPM3B_GFS_1.q_iRawPress <-> AI Standard Channel 3/GVL_SXR_VAC.fb_PCPM3B_GFS_1.i_iPRESS_R
//     SimTask Outputs/GVL_SXR_VAC.st_SL1K0_GCC_1.q_iRawPress <-> AI Standard Channel 1/GVL_SXR_VAC.fb_SL1K0_GCC_1.i_iPRESS_R
//     SimTask Outputs/GVL_SXR_VAC.st_SL1K0_GPI_1.q_iRawPress <-> AI Standard Channel 5/GVL_SXR_VAC.fb_SL1K0_GPI_1.i_iPRESS_R
//   plc_kfe_vac_sim/plc_kfe_vac_sim Instance <-> SimDevice 2 (EtherCAT Simulation)/=+-ES3068_01_05
//     SimTask Outputs/GVL_SXR_VAC.st_TV2K0_GCC_1.q_iRawPress <-> AI Standard Channel 1/GVL_SXR_VAC.fb_TV2K0_GCC_1.i_iPRESS_R
//     SimTask Outputs/GVL_SXR_VAC.st_TV2K0_GCC_2.q_iRawPress <-> AI Standard Channel 3/GVL_SXR_VAC.fb_TV2K0_GCC_2.i_iPRESS_R
//     SimTask Outputs/GVL_SXR_VAC.st_TV2K0_GPI_1.q_iRawPress <-> AI Standard Channel 5/GVL_SXR_VAC.fb_TV2K0_GPI_1.i_iPRESS_R
//     SimTask Outputs/GVL_SXR_VAC.st_TV2K0_GPI_2.q_iRawPress <-> AI Standard Channel 6/GVL_SXR_VAC.fb_TV2K0_GPI_2.i_iPRESS_R
//   plc_kfe_vac_sim/plc_kfe_vac_sim Instance <-> SimDevice 2 (EtherCAT Simulation)/=+-ES3068_01_08
//     SimTask Outputs/GVL_SXR_VAC.st_MR1K1_BEND_GCC_1.q_iRawPress <-> AI Standard Channel 3/GVL_SXR_VAC.fb_MR1K1_BEND_GCC_1.i_iPRESS_R
//     SimTask Outputs/GVL_SXR_VAC.st_MR1K1_BEND_GPI_1.q_iRawPress <-> AI Standard Channel 6/GVL_SXR_VAC.fb_MR1K1_BEND_GPI_1.i_iPRESS_R
//     SimTask Outputs/GVL_SXR_VAC.st_PA1K0_GCC_1.q_iRawPress <-> AI Standard Channel 1/GVL_SXR_VAC.fb_PA1K0_GCC_1.i_iPRESS_R
//     SimTask Outputs/GVL_SXR_VAC.st_PA1K0_GPI_1.q_iRawPress <-> AI Standard Channel 5/GVL_SXR_VAC.fb_PA1K0_GPI_1.i_iPRESS_R

CONFIGURATION plc_kfe_vac
    RESOURCE PLC ON TwinCAT3
        TASK FSV_task(INTERVAL := T#1ms, PRIORITY := 13);
        TASK PlcTask(INTERVAL := T#10ms, PRIORITY := 41);
        PROGRAM PRG_VFS WITH FSV_task : PRG_VFS;
        PROGRAM MAIN WITH PlcTask : MAIN;
    END_RESOURCE
END_CONFIGURATION

// ---- DUTs/ST_EXT_GCC.TcDUT
TYPE ST_EXT_GCC :
STRUCT
    {attribute 'pytmc' := '
        pv: ILK_INP;
        io: io;
    '}
    xIlk_Inp: BOOL; // Report the input signal .
END_STRUCT
END_TYPE

// ---- DUTs/ST_EXT_ILK.TcDUT
TYPE ST_EXT_ILK :
STRUCT
    {attribute 'pytmc' := '
    pv: HV_SW;
    io: io;
    '}
    xIlk_sw: BOOL:=True; // EPICS control for switching the interlock on or off.
    {attribute 'pytmc' := '
    pv: ILK_DO;
    io: i;
    '}
    q_xILK_OK_DO: BOOL; // Readout of the external interlock's ouput value
    {attribute 'pytmc' := '
    pv: ILK_OK;
    io: i;
    '}
    xIlkOK	:	BOOL := FALSE; // Interlock Bit
    {attribute 'pytmc' := '
    pv: PRO_SP;
    io: io;
    '}
    rPRO_SP: REAL	:= 1e-6; // Pressure below which the HV signal may turn on
END_STRUCT
END_TYPE

// ---- GVLs/GVL_SXR_VAC.TcGVL
VAR_GLOBAL


// FB_MKS317

{attribute 'pytmc' := ' pv: RTDSK0:GPI:1 '}
fb_RTDSK0_GPI_1 : FB_MKS317;
{attribute 'pytmc' := ' pv: IM1K0:XTES:GPI:1 '}
fb_IM1K0_XTES_GPI_1 : FB_MKS317;
{attribute 'pytmc' := ' pv: SL1K0:POWER:GPI:1 '}
fb_SL1K0_POWER_GPI_1 : FB_MKS317;
{attribute 'pytmc' := ' pv: TV2K0:GPI:1 '}
fb_TV2K0_GPI_1 : FB_MKS317;
{attribute 'pytmc' := ' pv: TV2K0:GPI:2 '}
fb_TV2K0_GPI_2 : FB_MKS317;
{attribute 'pytmc' := ' pv: PA1K0:GPI:1 '}
fb_PA1K0_GPI_1 : FB_MKS317;


// MKS275 Gauges

{attribute 'pytmc' := ' pv: MR1K1:BEND:GPI:1 '}
fb_MR1K1_BEND_GPI_1 : FB_MKS275;
{attribute 'pytmc' := ' pv: MR1K3:TXI:GPI:1 '}
fb_MR1K3_TXI_GPI_1 : FB_MKS275;
{attribute 'pytmc' := ' pv: MR2K3:TXI:GPI:1 '}
fb_MR2K3_TXI_GPI_1 : FB_MKS275;
{attribute 'pytmc' := ' pv: SP1K1:MONO:GPI:1 '}
fb_SP1K1_MONO_GPI_1 : FB_MKS275;
{attribute 'pytmc' := ' pv: TV3K0:GPI:1 '}
fb_TV3K0_GPI_1 : FB_MKS275;
{attribute 'pytmc' := ' pv: MR1K4:SOMS:GPI:1 '}
fb_MR1K4_SOMS_GPI_1 : FB_MKS275;


// FB_MKS422

{attribute 'pytmc' := ' pv: RTDSK0:GCC:1 '}
fb_RTDSK0_GCC_1 : FB_MKS422;
{attribute 'pytmc' := ' pv: IM1K0:XTES:GCC:1 '}
fb_IM1K0_XTES_GCC_1 : FB_MKS422;
{attribute 'pytmc' := ' pv: PCPM3B:GFS:1 '}
fb_PCPM3B_GFS_1 : FB_MKS422;
{attribute 'pytmc' := ' pv: SL1K0:POWER:GCC:1 '}
fb_SL1K0_POWER_GCC_1 : FB_MKS422;
{attribute 'pytmc' := ' pv: TV2K0:GCC:1 '}
fb_TV2K0_GCC_1 : FB_MKS422;
{attribute 'pytmc' := ' pv: TV2K0:GCC:2 '}
fb_TV2K0_GCC_2 : FB_MKS422;
{attribute 'pytmc' := ' pv: PA1K0:GCC:1 '}
fb_PA1K0_GCC_1 : FB_MKS422;



// MKS500_EP Gauges

{attribute 'pytmc' := ' pv: MR1K1:BEND:GCC:1 '}
fb_MR1K1_BEND_GCC_1 : FB_MKS500;
{attribute 'pytmc' := ' pv: MR1K3:TXI:GCC:1 '}
fb_MR1K3_TXI_GCC_1 : FB_MKS500;
{attribute 'pytmc' := ' pv: MR2K3:TXI:GCC:1 '}
fb_MR2K3_TXI_GCC_1 : FB_MKS500;
{attribute 'pytmc' := ' pv: SP1K1:MONO:GCC:1 '}
fb_SP1K1_MONO_GCC_1 : FB_MKS500;
{attribute 'pytmc' := ' pv: TV3K0:GCC:1 '}
fb_TV3K0_GCC_1 : FB_MKS500;
{attribute 'pytmc' := ' pv: MR1K4:SOMS:GCC:1 '}
fb_MR1K4_SOMS_GCC_1 : FB_MKS500;


// VGC Valves

{attribute 'pytmc' := ' pv: RTDSK0:VGC:1 '}
fb_RTDSK0_VGC_1 : FB_VGC;
{attribute 'pytmc' := ' pv: EM1K0:GMD:VGC:1 '}
fb_EM1K0_GMD_VGC_1 : FB_VGC;
{attribute 'pytmc' := ' pv: AT1K0:GAS:VGC:1 '}
fb_AT1K0_GAS_VGC_1 : FB_VGC;
{attribute 'pytmc' := ' pv: EM2K0:XGMD:VGC:1 '}
fb_EM2K0_XGMD_VGC_1 : FB_VGC;
{attribute 'pytmc' := ' pv: EM2K0:XGMD:VGC:2 '}
fb_EM2K0_XGMD_VGC_2 : FB_VGC;
{attribute 'pytmc' := ' pv: TV2K0:VGC:1 '}
fb_TV2K0_VGC_1 : FB_VGC;
{attribute 'pytmc' := ' pv: MR1K1:VGC:1 '}
fb_MR1K1_BEND_VGC_1 : FB_VGC;
{attribute 'pytmc' := ' pv: MR1K3:VGC:1 '}
fb_MR1K3_TXI_VGC_1 : FB_VGC;
{attribute 'pytmc' := ' pv: SP1K1:MONO:VGC:1 '}
fb_SP1K1_MONO_VGC_1 : FB_VGC;
{attribute 'pytmc' := ' pv: SP1K1:MONO:VGC:2 '}
fb_SP1K1_MONO_VGC_2 : FB_VGC;
{attribute 'pytmc' := ' pv: IM1K3:PPM:VGC:1 '}
fb_IM1K3_PPM_VGC_1 : FB_VGC;
{attribute 'pytmc' := ' pv: TV3K0:VGC:1 '}
fb_TV3K0_VGC_1 : FB_VGC;
{attribute 'pytmc' := ' pv: MR1K4:VGC:1 '}
fb_MR1K4_SOMS_VGC_1 : FB_VGC;
{attribute 'pytmc' := ' pv: IM1K0:XTES:VGC:1 '}
//linking pragma needed
{attribute 'TcLinkTo' := 	'.i_xOpnLS	:=	TIIB[=+-EL1004_03_04]^Channel 3^Input;
                            .i_xClsLS	:=	TIIB[=+-EL1004_03_04]^Channel 4^Input;
                            .q_xOPN_DO	:=	TIIB[=+-ES2004_03_03]^Channel 3^Output;
                            .q_xOPN_DO	:=	TIIB[=+-ES2004_03_03]^Channel 4^Output'}
fb_IM1K0_XTES_VGC_1 : FB_VGC;

// VFS valves

   {attribute 'TcLinkTo' := '.q_xPress_OK		:= 	TIPC^plc_kfe_vac_fs^plc_kfe_vac_fs Instance^PlcTask Inputs^GVL_SXR_VAC_FS_DEVICES.fb_TV2K0_VFS_1.i_xPress_OK;
                             .q_xOPN_SW			:=  TIPC^plc_kfe_vac_fs^plc_kfe_vac_fs Instance^PlcTask Inputs^GVL_SXR_VAC_FS_DEVICES.fb_TV2K0_VFS_1.i_xOPN_SW;
                             .q_xCLS_SW			:=  TIPC^plc_kfe_vac_fs^plc_kfe_vac_fs Instance^PlcTask Inputs^GVL_SXR_VAC_FS_DEVICES.fb_TV2K0_VFS_1.i_xCLS_SW;
                             .q_xVAC_FAULT_Reset:= 	TIPC^plc_kfe_vac_fs^plc_kfe_vac_fs Instance^PlcTask Inputs^GVL_SXR_VAC_FS_DEVICES.fb_TV2K0_VFS_1.i_xVAC_FAULT_Reset;
                             .q_xOverrideMode	:= 	TIPC^plc_kfe_vac_fs^plc_kfe_vac_fs Instance^PlcTask Inputs^GVL_SXR_VAC_FS_DEVICES.fb_TV2K0_VFS_1.i_xOverrideMode;
                             .q_xOverrideOpen	:= 	TIPC^plc_kfe_vac_fs^plc_kfe_vac_fs Instance^PlcTask Inputs^GVL_SXR_VAC_FS_DEVICES.fb_TV2K0_VFS_1.i_xOverrideOpen;
                             .i_xTrigger		:=	TIPC^plc_kfe_vac_fs^plc_kfe_vac_fs Instance^PlcTask Outputs^GVL_SXR_VAC_FS_DEVICES.fb_TV2K0_VFS_1.q_xTrigger;
                             .i_xVFS_Open		:=	TIPC^plc_kfe_vac_fs^plc_kfe_vac_fs Instance^PlcTask Outputs^GVL_SXR_VAC_FS_DEVICES.fb_TV2K0_VFS_1.q_xVFS_Open;
                             .i_xVFS_Closed		:=	TIPC^plc_kfe_vac_fs^plc_kfe_vac_fs Instance^PlcTask Outputs^GVL_SXR_VAC_FS_DEVICES.fb_TV2K0_VFS_1.q_xVFS_Closed;
                             .i_xVAC_FAULT_OK	:=	TIPC^plc_kfe_vac_fs^plc_kfe_vac_fs Instance^PlcTask Outputs^GVL_SXR_VAC_FS_DEVICES.fb_TV2K0_VFS_1.q_xVAC_FAULT_OK;
                             .i_xMPS_OK			:=  TIPC^plc_kfe_vac_fs^plc_kfe_vac_fs Instance^PlcTask Outputs^GVL_SXR_VAC_FS_DEVICES.fb_TV2K0_VFS_1.q_xMPS_OK;
                             .i_eVFS_State		:=	TIPC^plc_kfe_vac_fs^plc_kfe_vac_fs Instance^PlcTask Outputs^GVL_SXR_VAC_FS_DEVICES.fb_TV2K0_VFS_1.q_eVFS_State
'}
{attribute 'pytmc' := '
    pv: TV2K0:VFS:1
    io: io
'}
fb_TV2K0_VFS_1_Interface : FB_VFS_Interface;


// PIP_Gamma Pumps

{attribute 'pytmc' := ' pv: RTDSK0:PIP:1 '}
fb_RTDSK0_PIP_1 : FB_PIP_GAMMA;
{attribute 'pytmc' := ' pv: RTDSK0:PIP:2 '}
fb_RTDSK0_PIP_2 : FB_PIP_GAMMA;
{attribute 'pytmc' := ' pv: RTDSK0:PIP:3 '}
fb_RTDSK0_PIP_3 : FB_PIP_GAMMA;
{attribute 'pytmc' := ' pv: RTDSK0:PIP:4 '}
fb_RTDSK0_PIP_4 : FB_PIP_GAMMA;
{attribute 'pytmc' := ' pv: RTDSK0:PIP:5 '}
fb_RTDSK0_PIP_5 : FB_PIP_GAMMA;
{attribute 'pytmc' := ' pv: PCPM3B:PIP:1 '}
fb_PCPM3B_PIP_1 : FB_PIP_GAMMA;
{attribute 'pytmc' := ' pv: PA1K0:PIP:1 '}
fb_PA1K0_PIP_1 : FB_PIP_GAMMA;
{attribute 'pytmc' := ' pv: PA1K0 '}
fb_PA1K0 : FB_PIP_GAMMA;
{attribute 'pytmc' := ' pv: MR1K1:BEND:PIP:1 '}
fb_MR1K1_BEND_PIP_1 : FB_PIP_GAMMA;
{attribute 'pytmc' := ' pv: MR1K3:TXI:PIP:1 '}
fb_MR1K3_TXI_PIP_1 : FB_PIP_GAMMA;
{attribute 'pytmc' := ' pv: MR2K3:TXI:PIP:1 '}
fb_MR2K3_TXI_PIP_1 : FB_PIP_GAMMA;
{attribute 'pytmc' := ' pv: SP1K1:MONO:PIP:1 '}
fb_SP1K1_MONO_PIP_1 : FB_PIP_GAMMA;
{attribute 'pytmc' := ' pv: SP1K1:MONO:PIP:2 '}
fb_SP1K1_MONO_PIP_2 : FB_PIP_GAMMA;
{attribute 'pytmc' := ' pv: TV3K0:PIP:1 '}
fb_TV3K0_PIP_1 : FB_PIP_GAMMA;
{attribute 'TcLinkTo' := 	'.i_iPRESS		:=	TIIB[=+-EL3064_02_07]^AI Standard Channel 1^Value;
                                 .i_xSP_DI		:= 	TIIB[=+-EL1004_02_09]^Channel 1^Input;
                                 .q_xHVEna_DO	:= 	TIIB[=+-EL2794_02_08]^Channel 1^Output
    '}
{attribute 'pytmc' := 'pv: SL1K0:POWER:PIP:01	'}
fb_SL1K0_PIP_1 : FB_PIP_GAMMA;





END_VAR

// ---- GVLs/GVL_VAC_INTF.TcGVL
VAR_GLOBAL

    // AD Interface
    {attribute 'pytmc' := ' pv: TV1K0:INTF:GCC:1 '}
    fb_TV1K0_INTF_GCC_1 : FB_EXT_TREATY_GAUGE;
    {attribute 'pytmc' := ' pv: RTDSK0:INTF:VGC:1 '}
    fb_RTDSK0_INTF_VGC_1 : FB_EXT_TREATY_VGC;


    // TMO vacuum interface
    {attribute 'pytmc' :=' pv: MR1K4:SOMS:GCC:1:ILK_UPPER'}
    st_TMO_ILK_Upper			:	ST_EXT_ILK;
    {attribute 'pytmc' :=' pv: MR1K4:SOMS:GCC:1:ILK_LOWER'}
    st_TMO_ILK_Lower			:	ST_EXT_ILK;

    fb_TMO_ILK_Uppper			:	FB_EXT_ILK;
    fb_TMO_ILK_Lower			:	FB_EXT_ILK;


    // RIX Interface
    {attribute 'pytmc' := ' pv: PC1K1:INTF:GCC:1 '}
    fb_PC1K1_INTF_GCC_1 : FB_EXT_TREATY_GAUGE;

     // TXI Interface
    {attribute 'pytmc' := ' pv: PC1K1:INTF:PIP:1 '}
    {attribute 'TcLinkTo' := 	'.i_xEXT_Press_OK		:=	TIIB[=+-ES1008_02_03]^Channel 3^Input;
    '}

    fb_PC1K3_INTF_PIP_1 : FB_EXT_TREATY_GAUGE;


    // EM1K0-GMD Vacuum Interface
    n_EM1K0_VAC_counter         :   UDINT;
    fb_EM1K0_GMD_GCC_10_reader  :   FB_TGCC_ADS;
    fb_EM1K0_GMD_GCC_70_reader  :   FB_TGCC_ADS;


    // AT1K0-GAS Vacuum Interface
    n_AT1K0_VAC_counter         :   UDINT;
    fb_AT1K0_GAS_GCC_10_reader  :   FB_TGCC_ADS;
    fb_AT1K0_GAS_GCC_140_reader :   FB_TGCC_ADS;


    // EM2K0-XGMD Vacuum Interface
    n_EM2K0_VAC_counter         :   UDINT;
    fb_EM2K0_XGMD_GCC_10_reader :   FB_TGCC_ADS;
    fb_EM2K0_XGMD_GCC_90_reader :   FB_TGCC_ADS;


END_VAR

// ---- GVLs/GVL_Variables.TcGVL
VAR_GLOBAL

// *******************
// Interlock overrides
// *******************

{attribute 'pytmc' := '
    pv: @(PREFIX)SYSOVERRIDE
'}
xSystemOverrideMode : BOOL; (* Global system override for the prototype section*)


// ***************************
// Hardware Fast fault outputs
// ***************************

// K0/SXR upstream specific faults
{attribute 'pytmc' := '
    pv: @(PREFIX)FFO:01
'}
g_FastFaultOutputK0  :   FB_HardwareFFOutput :=(i_sNetID:='172.21.92.73.1.1');

// K2/RIX specific faults
{attribute 'pytmc' := '
    pv: @(PREFIX)FFO:02
'}
g_FastFaultOutputK2  :   FB_HardwareFFOutput :=(i_sNetID:='172.21.92.73.1.1');

// K3/TXI specific faults
{attribute 'pytmc' := '
    pv: @(PREFIX)FFO:03
'}
g_FastFaultOutputK3  :   FB_HardwareFFOutput :=(i_sNetID:='172.21.92.73.1.1');

// K4/TMO specific faults
{attribute 'pytmc' := '
    pv: @(PREFIX)FFO:04
'}
g_FastFaultOutputK4  :   FB_HardwareFFOutput :=(i_sNetID:='172.21.92.73.1.1');

// Fault aggregator for combined beamline
{attribute 'TcLinkTo' := '.q_xFastFaultOut:=TIIB[PMPS_FFO (EL2202)]^Channel 1^Output'}
g_FastFaultOutputAll  :   FB_HardwareFFOutput :=(i_sNetID:='172.21.92.73.1.1');

{attribute 'pytmc' := '
    pv: @(PREFIX)FFO:05
'}
{attribute 'TcLinkTo' := '.q_xFastFaultOut:=TIIB[PMPS_FFO (EL2202)]^Channel 2^Output'}
g_FastFaultOutput2  :	FB_HardwareFFOutput :=(i_sNetID:='172.21.92.73.1.1');	//FFO for Fast Shutter Valves upstream of ST1L0_XTES


// Dummy FFO for valves not yet allowed to open. To be removed when proper interfaces to TXI and RIX vacuum are implemented.
{attribute 'pytmc' := '
    pv: @(PREFIX)FF1A
'}
g_FastFaultOutputINTF  :   FB_HardwareFFOutput :=(i_sNetID:='172.21.92.73.1.1');


// ************
// FB_FastFault
// ************

g_FastFault		:	FB_FastFault;


// *****************
// Fast fault resets
// *****************

{attribute 'pytmc' := '
pv: @(PREFIX)RESET:FF1
'}
xReset_PMPS_FFO_K0	:	BOOL	:=	FALSE;

{attribute 'pytmc' := '
pv: @(PREFIX)RESET:FF2
'}
xReset_PMPS_FFO_K2	:	BOOL	:=	FALSE;

{attribute 'pytmc' := '
pv: @(PREFIX)RESET:FF3
'}
xReset_PMPS_FFO_K3	:	BOOL	:=	FALSE;

{attribute 'pytmc' := '
pv: @(PREFIX)RESET:FF4
'}
xReset_PMPS_FFO_K4	:	BOOL	:=	FALSE;


// *******
// Logging
// *******

fbLogHandler : FB_loghandler;
fbEcatDiagWrapper : FB_EcatDiagWrapper;


// *******
// Arbiter
// *******

{attribute 'pytmc' := '
     pv: @(PREFIX)Arb:01
'}
g_fbArbiter1    :   FB_Arbiter(01);


END_VAR

// ---- GVLs/GVL_VFS.TcGVL
VAR_GLOBAL

//Fast Shutter
   {attribute 'pytmc' := '
        pv: TV2K0:VFS:1
    '}
    {attribute 'TcLinkTo' := 	'
        .q_xClose_A	:=	TIID^Device 1 (EtherCAT)^=+-EK1100_05_01^=+-ES2202_05_03^Channel 1^GVL_SXR_VAC_FS_DEVICES.fb_TV2K0_VFS_1.q_xClose_A;
        .q_xClose_B	:=	TIID^Device 1 (EtherCAT)^=+-EK1100_05_01^=+-ES2202_05_03^Channel 2^GVL_SXR_VAC_FS_DEVICES.fb_TV2K0_VFS_1.q_xClose_B;
        .q_xClose_C	:=	TIID^Device 1 (EtherCAT)^=+-EK1100_05_01^=+-ES2202_05_04^Channel 1^GVL_SXR_VAC_FS_DEVICES.fb_TV2K0_VFS_1.q_xClose_C;
        .q_xOPN_DO	:=	TIID^Device 1 (EtherCAT)^=+-EK1100_05_01^=+-ES2202_05_04^Channel 2^GVL_SXR_VAC_FS_DEVICES.fb_TV2K0_VFS_1.q_xOPN_DO;
        .i_xClsLS	:=	TIID^Device 1 (EtherCAT)^=+-EK1100_05_01^=+-ES1004_05_02^Channel 1^GVL_SXR_VAC_FS_DEVICES.fb_TV2K0_VFS_1.i_xClsLS;
        .i_xOpnLS	:=	TIID^Device 1 (EtherCAT)^=+-EK1100_05_01^=+-ES1004_05_02^Channel 2^GVL_SXR_VAC_FS_DEVICES.fb_TV2K0_VFS_1.i_xOpnLS;
        .i_xTrigger :=  TIID^Device 1 (EtherCAT)^=+-EK1100_02_00^=+-EL1124_02_11^Channel 1^GVL_SXR_VAC_FS_DEVICES.fb_TV2K0_VFS_1.i_xTrigger;
        .i_xPress_OK		:= 	TIPC^plc_kfe_vac^plc_kfe_vac Instance^PlcTask Outputs^GVL_SXR_VAC.fb_TV2K0_VFS_1_Interface.q_xPRESS_OK;
        .i_xOPN_SW			:=  TIPC^plc_kfe_vac^plc_kfe_vac Instance^PlcTask Outputs^GVL_SXR_VAC.fb_TV2K0_VFS_1_Interface.q_xOPN_SW;
        .i_xCLS_SW			:=  TIPC^plc_kfe_vac^plc_kfe_vac Instance^PlcTask Outputs^GVL_SXR_VAC.fb_TV2K0_VFS_1_Interface.q_xCLS_SW;
        .i_xVAC_FAULT_Reset:= 	TIPC^plc_kfe_vac^plc_kfe_vac Instance^PlcTask Outputs^GVL_SXR_VAC.fb_TV2K0_VFS_1_Interface.q_xVAC_FAULT_Reset;
        .i_xOverrideMode	:= 	TIPC^plc_kfe_vac^plc_kfe_vac Instance^PlcTask Outputs^GVL_SXR_VAC.fb_TV2K0_VFS_1_Interface.q_xOverrideMode;
        .i_xOverrideOpen	:= 	TIPC^plc_kfe_vac^plc_kfe_vac Instance^PlcTask Outputs^GVL_SXR_VAC.fb_TV2K0_VFS_1_Interface.q_xOverrideOpen;
        .q_xTrigger		:=	TIPC^plc_kfe_vac^plc_kfe_vac Instance^PlcTask Inputs^GVL_SXR_VAC.fb_TV2K0_VFS_1_Interface.i_xTrigger;
        .q_xVFS_Open		:=	TIPC^plc_kfe_vac^plc_kfe_vac Instance^PlcTask Inputs^GVL_SXR_VAC.fb_TV2K0_VFS_1_Interface.i_xVFS_Open;
        .q_xVFS_Closed		:=	TIPC^plc_kfe_vac^plc_kfe_vac Instance^PlcTask Inputs^GVL_SXR_VAC.fb_TV2K0_VFS_1_Interface.i_xVFS_Closed;
        .q_xVAC_FAULT_OK	:= TIPC^plc_kfe_vac^plc_kfe_vac Instance^PlcTask Inputs^GVL_SXR_VAC.fb_TV2K0_VFS_1_Interface.i_xVAC_FAULT_OK;
        .q_xMPS_OK			:=  TIPC^plc_kfe_vac^plc_kfe_vac Instance^PlcTask Inputs^GVL_SXR_VAC.fb_TV2K0_VFS_1_Interface.i_xMPS_OK;
        .q_eVFS_State		:=	TIPC^plc_kfe_vac^plc_kfe_vac Instance^PlcTask Inputs^GVL_SXR_VAC.fb_TV2K0_VFS_1_Interface.i_eVFS_State;
        .i_xVetoValveOpenDO := ;
        .i_xVetoValveClosed :=
    '}
    fb_TV2K0_VFS_1 : FB_VFS;

END_VAR

// ---- POUs/PRG_VFS.TcPOU
PROGRAM PRG_VFS
VAR
END_VAR

fb_TV2K0_VFS_1(
    i_xPMPS_OK:= TRUE,
    i_xExt_OK:= TRUE,
    i_sDevName:= 'TV2K0:VFS:1',
    io_fbFFHWO:= g_FastFaultOutput2
);

(*FastFaultOuput*)
g_FastFaultOutput2.Execute(bAutoReset:= TRUE);

END_PROGRAM

// ---- POUs/MAIN.TcPOU
PROGRAM MAIN
VAR

    fbGetCurTaskIdx  : GETCURTASKINDEX;
//	tRecover_pip: TON;
//	tRecover_gcc: TON;
//	bRecover_pip : BOOL ;
//	bRecover_gcc : BOOL ;
    // For Persistent Data
    fbWritePersistentData           : WritePersistentData;
//	tWait_pip:TIME:=T#900S;
//	tWait_gcc:TIME:=T#600S;

END_VAR

PRG_DIAGNOSTIC();
PRG_SXR_VAC();
PRG_VAC_INTF();
PRG_PMPS();
fbEcatDiagWrapper();
fbLogHandler();

(*
(* Auto Recover Ion pumps and vacuum cold cathode gauges after power outage*)
fbWritePersistentData(NETID:='', PORT:=851, START:=TRUE, TMOUT:=T#1s );

IF (bRecoverEnable) THEN

ACT_Recover();

END_IF
*)

END_PROGRAM

// ---- POUs/PRG_DIAGNOSTIC.TcPOU
PROGRAM PRG_DIAGNOSTIC
VAR

   fbTime : FB_LocalSystemTime := ( bEnable := TRUE, dwCycle := 1 );
   logTimer : TON := ( IN := TRUE, PT := T#1000ms );

   plcName : STRING[15];

   {attribute 'pytmc' := ' pv: simHeartbeat '}
   simHeartbeat AT %I* : UINT := 0;
   {attribute 'pytmc' := ' pv: plcHeartbeat '}
   plcHeartbeat : UDINT := 0;
   {attribute 'pytmc' := ' pv: plcInfo '}
   plcInfo : STRING[40];
   {attribute 'pytmc' := ' pv: plcLocalTime '}
   plcLocalTime : STRING[25];

END_VAR

plcHeartbeat := plcHeartbeat + 1;
IF plcHeartbeat > 4294967000
   THEN plcHeartbeat := 0;
END_IF

// get timestamp as string every second
fbTime();
logTimer( IN := fbTime.bValid );
IF logTimer.Q THEN
   logTimer( IN := FALSE ); logTimer( IN := fbTime.bValid );
   plcLocalTime := SYSTEMTIME_TO_STRING(fbTime.systemTime);
END_IF

// make an info string
plcName := 'Prototype PLC: ';
plcInfo := CONCAT(plcName, plcLocalTime);

END_PROGRAM

// ---- POUs/PRG_SXR_VAC.TcPOU
PROGRAM PRG_SXR_VAC
VAR
END_VAR




// MKS275 Gauges

fb_MR1K1_BEND_GPI_1(PG=>);
fb_MR2K3_TXI_GPI_1(PG=>);
fb_MR1K3_TXI_GPI_1(PG=>);
fb_SP1K1_MONO_GPI_1(PG=>);
fb_TV3K0_GPI_1(PG=>);
fb_MR1K4_SOMS_GPI_1(PG=>);

// MKS500_EP Gauges

fb_MR1K1_BEND_GCC_1(PG := fb_MR1K1_BEND_GPI_1.PG, bEP:=TRUE);
fb_MR2K3_TXI_GCC_1(PG := fb_MR2K3_TXI_GPI_1.PG, bEP:=TRUE);
fb_MR1K3_TXI_GCC_1(PG := fb_MR1K3_TXI_GPI_1.PG, bEP:=TRUE);
fb_SP1K1_MONO_GCC_1(PG := fb_SP1K1_MONO_GPI_1.PG, bEP:=TRUE);
fb_TV3K0_GCC_1(PG := fb_TV3K0_GPI_1.PG, bEP:=TRUE);
fb_MR1K4_SOMS_GCC_1(PG := fb_MR1K4_SOMS_GPI_1.PG, bEP:=TRUE);

// VGC Valves

fb_RTDSK0_VGC_1( i_stUSG := fb_TV1K0_INTF_GCC_1.IG, i_stDSG := fb_RTDSK0_GCC_1.IG, i_xDis_DPIlk := FALSE,
                i_xEPS_OK := TRUE, i_xPMPS_OK := TRUE, i_xExt_OK := TRUE, i_xOverrideMode := xSystemOverrideMode,
                i_xReset := xReset_PMPS_FFO_K0, io_fbFFHWO := g_FastFaultOutputK0, fbArbiter := g_fbArbiter1 ,
                i_sDevName := 'RTDSK0:VGC:1' );

fb_EM1K0_GMD_VGC_1(i_stUSG := fb_RTDSK0_GCC_1.IG, i_stDSG := fb_EM1K0_GMD_GCC_10_reader.IG, i_xDis_DPIlk := FALSE,
                i_xEPS_OK := TRUE, i_xPMPS_OK := TRUE, i_xExt_OK := (NOT fb_EM1K0_GMD_GCC_10_reader.bError),
                   i_xOverrideMode := xSystemOverrideMode, i_xReset := xReset_PMPS_FFO_K0, io_fbFFHWO := g_FastFaultOutputK0,
                fbArbiter := g_fbArbiter1,  i_sDevName := 'EM1K0:GMD:VGC:1');

fb_AT1K0_GAS_VGC_1(i_stUSG := fb_PCPM3B_PIP_1.q_IG, i_stDSG := fb_AT1K0_GAS_GCC_10_reader.IG, i_xDis_DPIlk := FALSE, i_xEPS_OK := TRUE, i_xPMPS_OK := TRUE,
                i_xExt_OK := (NOT fb_AT1K0_GAS_GCC_10_reader.bError), i_xOverrideMode := xSystemOverrideMode,
                i_xReset := xReset_PMPS_FFO_K0, io_fbFFHWO := g_FastFaultOutputK0, fbArbiter := g_fbArbiter1, i_sDevName := 'AT1K0:GAS:VGC:1' );

fb_EM2K0_XGMD_VGC_1(i_stUSG := fb_AT1K0_GAS_GCC_140_reader.IG, i_stDSG := fb_EM2K0_XGMD_GCC_10_reader.IG, i_xDis_DPIlk := FALSE, i_xEPS_OK := TRUE, i_xPMPS_OK := TRUE,
                i_xExt_OK := (NOT fb_AT1K0_GAS_GCC_140_reader.bError) AND (NOT fb_EM2K0_XGMD_GCC_10_reader.bError),
                i_xOverrideMode := xSystemOverrideMode, i_xReset := xReset_PMPS_FFO_K0, io_fbFFHWO := g_FastFaultOutputK0, fbArbiter := g_fbArbiter1, i_sDevName := 'EM2K0:XGMD:VGC:1');

fb_EM2K0_XGMD_VGC_2(i_stUSG := fb_EM2K0_XGMD_GCC_90_reader.IG, i_stDSG := fb_TV2K0_GCC_1.IG, i_xDis_DPIlk := FALSE, i_xEPS_OK := TRUE, i_xPMPS_OK := TRUE,
                i_xExt_OK := (NOT fb_EM2K0_XGMD_GCC_90_reader.bError), i_xOverrideMode := xSystemOverrideMode,
                i_xReset := xReset_PMPS_FFO_K0, io_fbFFHWO := g_FastFaultOutputK0, fbArbiter := g_fbArbiter1, i_sDevName := 'EM2K0:XGMD:VGC:2');

fb_TV2K0_VGC_1(i_stUSG := fb_TV2K0_GCC_1.IG, i_stDSG := fb_TV2K0_GCC_2.IG, i_xDis_DPIlk := FALSE, i_xEPS_OK := TRUE,
                 i_xPMPS_OK := TRUE, i_xExt_OK := fb_TV2K0_VFS_1_Interface.i_xVAC_FAULT_OK, i_xOverrideMode := xSystemOverrideMode, i_xReset := xReset_PMPS_FFO_K0,
                io_fbFFHWO := g_FastFaultOutputK0, fbArbiter := g_fbArbiter1, i_sDevName := 'TV2K0:VGC:1');

fb_MR1K1_BEND_VGC_1(i_stUSG :=  fb_PA1K0.q_IG, i_stDSG :=fb_MR1K1_BEND_PIP_1.q_IG, i_xDis_DPIlk := FALSE, i_xEPS_OK := TRUE, i_xPMPS_OK := TRUE,
                i_xExt_OK := fb_TV2K0_VFS_1_Interface.i_xVAC_FAULT_OK, i_xOverrideMode := xSystemOverrideMode, i_xReset := xReset_PMPS_FFO_K0,
                io_fbFFHWO := g_FastFaultOutputK0, fbArbiter := g_fbArbiter1,i_sDevName := 'MR1K1:BEND:VGC:1');

fb_MR1K3_TXI_VGC_1(i_stUSG := fb_MR1K1_BEND_PIP_1.q_IG, i_stDSG := fb_MR1K3_TXI_PIP_1.q_IG, i_xDis_DPIlk := FALSE, i_xEPS_OK := TRUE,
                i_xPMPS_OK := TRUE, i_xExt_OK := TRUE, i_xOverrideMode := xSystemOverrideMode, i_xReset := xReset_PMPS_FFO_K0,
                io_fbFFHWO := g_FastFaultOutputK0, fbArbiter := g_fbArbiter1, i_sDevName := 'MR1K3:TXI:VGC:1');

fb_SP1K1_MONO_VGC_1(i_stUSG := fb_MR2K3_TXI_PIP_1.q_IG, i_stDSG := fb_SP1K1_MONO_PIP_1.q_IG, i_xDis_DPIlk := FALSE,
                i_xEPS_OK := TRUE, i_xPMPS_OK := TRUE, i_xExt_OK := TRUE, i_xOverrideMode := xSystemOverrideMode,
                i_xReset := xReset_PMPS_FFO_K2, io_fbFFHWO := g_FastFaultOutputK2, fbArbiter := g_fbArbiter1, i_sDevName := 'SP1K1:MONO:VGC:1');

fb_SP1K1_MONO_VGC_2(i_stUSG := fb_SP1K1_MONO_PIP_1.q_IG, i_stDSG := fb_PC1K1_INTF_GCC_1.IG, i_xDis_DPIlk := FALSE,
                i_xEPS_OK := TRUE, i_xPMPS_OK := TRUE, i_xExt_OK := TRUE, i_xOverrideMode := xSystemOverrideMode,
                i_xReset := xReset_PMPS_FFO_K2, io_fbFFHWO := g_FastFaultOutputK2, fbArbiter := g_fbArbiter1, i_sDevName := 'SP1K1:MONO:VGC:2');

fb_IM1K3_PPM_VGC_1(i_stUSG := fb_MR2K3_TXI_PIP_1.q_IG, i_stDSG := , i_xDis_DPIlk := FALSE, i_xEPS_OK := TRUE, i_xPMPS_OK := TRUE,
                i_xExt_OK := TRUE, i_xOverrideMode := xSystemOverrideMode, i_xReset := xReset_PMPS_FFO_K3, io_fbFFHWO := g_FastFaultOutputK3,
                fbArbiter := g_fbArbiter1, i_sDevName := 'IM1K3:PPM:VGC:1');

fb_TV3K0_VGC_1(i_stUSG := fb_MR2K3_TXI_PIP_1.q_IG, i_stDSG := fb_TV3K0_PIP_1.q_IG, i_xDis_DPIlk := FALSE, i_xEPS_OK := TRUE,
                i_xPMPS_OK := TRUE, i_xExt_OK := TRUE, i_xOverrideMode := xSystemOverrideMode, i_xReset := xReset_PMPS_FFO_K4,
                io_fbFFHWO := g_FastFaultOutputK4, fbArbiter := g_fbArbiter1, i_sDevName := 'TV3K0:VGC:1');

fb_MR1K4_SOMS_VGC_1(i_stUSG := fb_TV3K0_PIP_1.q_IG, i_stDSG := fb_MR1K4_SOMS_GCC_1.IG, i_xDis_DPIlk := FALSE, i_xEPS_OK := TRUE,
                i_xPMPS_OK := TRUE, i_xExt_OK := TRUE, i_xOverrideMode := xSystemOverrideMode, i_xReset := xReset_PMPS_FFO_K4, io_fbFFHWO := g_FastFaultOutputK4,
                fbArbiter := g_fbArbiter1, i_sDevName := 'MR1K4:SOMS:VGC:1');

fb_IM1K0_XTES_VGC_1(i_stUSG := fb_IM1K0_XTES_GCC_1.IG, i_stDSG := fb_PCPM3B_PIP_1.q_IG, i_xDis_DPIlk := FALSE, i_xEPS_OK := TRUE,
                i_xPMPS_OK := TRUE, i_xExt_OK := TRUE, i_xOverrideMode := xSystemOverrideMode, i_xReset := xReset_PMPS_FFO_K0,
                io_fbFFHWO := g_FastFaultOutputK0, fbArbiter := g_fbArbiter1, i_sDevName :='IM1K0:XTES:VGC:1');

// VFS Valves

fb_TV2K0_VFS_1_Interface(IG := fb_PCPM3B_GFS_1.IG);

// PIP_Gamma Pumps

fb_RTDSK0_PIP_1(	i_stGauge := fb_RTDSK0_GCC_1.IG,		i_xOverrideMode := xSystemOverrideMode);
fb_RTDSK0_PIP_2(	i_stGauge := fb_RTDSK0_GCC_1.IG,		i_xOverrideMode := xSystemOverrideMode);
fb_RTDSK0_PIP_3(	i_stGauge := fb_RTDSK0_GCC_1.IG,		i_xOverrideMode := xSystemOverrideMode);
fb_RTDSK0_PIP_4(	i_stGauge := fb_RTDSK0_GCC_1.IG,		i_xOverrideMode := xSystemOverrideMode);
fb_RTDSK0_PIP_5(	i_stGauge := fb_RTDSK0_GCC_1.IG,		i_xOverrideMode := xSystemOverrideMode);
fb_PCPM3B_PIP_1(	i_stGauge := fb_PCPM3B_GFS_1.IG,		i_xOverrideMode := xSystemOverrideMode);
fb_PA1K0_PIP_1(		i_stGauge := fb_PA1K0_GCC_1.IG,			i_xOverrideMode := xSystemOverrideMode);
fb_PA1K0(			i_stGauge := fb_PA1K0_GCC_1.IG,			i_xOverrideMode := xSystemOverrideMode);
fb_MR1K1_BEND_PIP_1(i_stGauge := fb_MR1K1_BEND_GPI_1.PG,	i_xOverrideMode := xSystemOverrideMode);
fb_MR1K3_TXI_PIP_1(	i_stGauge := fb_MR1K3_TXI_GCC_1.IG,		i_xOverrideMode := xSystemOverrideMode);
fb_MR2K3_TXI_PIP_1(	i_stGauge := fb_MR1K3_TXI_GCC_1.IG,		i_xOverrideMode := xSystemOverrideMode);
fb_SP1K1_MONO_PIP_1(i_stGauge := fb_SP1K1_MONO_GPI_1.PG,	i_xOverrideMode := xSystemOverrideMode);
fb_SP1K1_MONO_PIP_2(i_stGauge := fb_SP1K1_MONO_GPI_1.PG,	i_xOverrideMode := xSystemOverrideMode);
fb_TV3K0_PIP_1(		i_stGauge := fb_TV3K0_GCC_1.IG,			i_xOverrideMode := xSystemOverrideMode);
fb_SL1K0_PIP_1( 	i_stGauge := fb_SL1K0_POWER_GPI_1.PG,	i_xOverrideMode := xSystemOverrideMode); // New Ion Pump



// FB_MKS422

fb_RTDSK0_GCC_1(PG := fb_RTDSK0_GPI_1.PG);
fb_IM1K0_XTES_GCC_1(PG := fb_IM1K0_XTES_GPI_1.PG);
fb_PCPM3B_GFS_1(PG := fb_SL1K0_POWER_GPI_1.PG);
fb_SL1K0_POWER_GCC_1(PG := fb_SL1K0_POWER_GPI_1.PG);
fb_TV2K0_GCC_1(PG := fb_TV2K0_GPI_1.PG);
fb_TV2K0_GCC_2(PG := fb_TV2K0_GPI_2.PG);
fb_PA1K0_GCC_1(PG := fb_PA1K0_GPI_1.PG);

// FB_MKS317

fb_RTDSK0_GPI_1(PG=>);
fb_IM1K0_XTES_GPI_1(PG=>);
fb_SL1K0_POWER_GPI_1(PG=>);
fb_TV2K0_GPI_1(PG=>);
fb_TV2K0_GPI_2(PG=>);
fb_PA1K0_GPI_1(PG=>);

END_PROGRAM

// ---- POUs/PRG_VAC_INTF.TcPOU
PROGRAM PRG_VAC_INTF
(*
This PRG governs the interfaces between the SXR Vacuum system and external systems.
This includes AD's vacuum system, EM1K0-GMD, AT1K0-GAS, EM2K0-XGMD, the TMO beamline vacuum system, and the RIX Beamline Vacuum System.
The Vacuum system for TXI is planned but not yet implemented. When implemented it should go here.
*)
VAR
END_VAR

// Interface to AD's vacuum system

fb_TV1K0_INTF_GCC_1(rTREATY_SIGNAL_PRESS := 5E-6, rNO_SIGNAL_PRESS := 760);
fb_RTDSK0_INTF_VGC_1(TREATY_VGC := fb_RTDSK0_VGC_1.iq_stValve);


// Update interlock signals for TMO
st_TMO_ILK_Upper.rPRO_SP 	:=	1E-4; // Fix the agreed-upon values
fb_TMO_ILK_Uppper(
    VG	:=	fb_MR1K4_SOMS_GCC_1.IG,
    ILK	:=	st_TMO_ILK_Upper
);
st_TMO_ILK_Lower.rPRO_SP	:=	1E-7; // Fix the agreed-upon values
fb_TMO_ILK_Lower(
    VG	:=	fb_MR1K4_SOMS_GCC_1.IG,
    ILK	:=	st_TMO_ILK_Lower
);


// Interface to RIX's vacuum system

fb_PC1K1_INTF_GCC_1(rTREATY_SIGNAL_PRESS := 5E-6, rNO_SIGNAL_PRESS := 760);

// Interface to TXI's K3 vacuum system

fb_PC1K3_INTF_PIP_1(rTREATY_SIGNAL_PRESS := 5E-6, rNO_SIGNAL_PRESS := 760);


// EM1K0-GMD Vacuum Interface

fb_EM1K0_GMD_GCC_10_reader(
    sNetId      :=  '172.21.92.59.1.1',
    nPort       :=  851,
    sVarName    :=  'GVL_GMD.fb_EM1K0_GMD_GCC_10',
    iWatchdog   :=  n_EM1K0_VAC_counter
);

fb_EM1K0_GMD_GCC_70_reader(
    sNetId      :=  '172.21.92.59.1.1',
    nPort       :=  851,
    sVarName    :=  'GVL_GMD.fb_EM1K0_GMD_GCC_70',
    iWatchdog   :=  n_EM1K0_VAC_counter
);


// AT1K0-GAS Vacuum Interface

fb_AT1K0_GAS_GCC_10_reader(
    sNetId      :=  '172.21.92.57.1.1',
    nPort       :=  851,
    sVarName    :=  'GVL_Devices.fb_AT1K0_GAS_GCC_10',
    iWatchdog   :=  n_AT1K0_VAC_counter
);

fb_AT1K0_GAS_GCC_140_reader(
    sNetId      :=  '172.21.92.57.1.1',
    nPort       :=  851,
    sVarName    :=  'GVL_Devices.fb_AT1K0_GAS_GCC_140',
    iWatchdog   :=  n_AT1K0_VAC_counter
);


// EM2K0-XGMD Vacuum Interface

fb_EM2K0_XGMD_GCC_10_reader(
    sNetId      :=  '172.21.92.60.1.1',
    nPort       :=  851,
    sVarName    :=  'GVL_GMD.fb_EM2K0_XGMD_GCC_10',
    iWatchdog   :=  n_EM2K0_VAC_counter
);

fb_EM2K0_XGMD_GCC_90_reader(
    sNetId      :=  '172.21.92.60.1.1',
    nPort       :=  851,
    sVarName    :=  'GVL_GMD.fb_EM2K0_XGMD_GCC_90',
    iWatchdog   :=  n_EM2K0_VAC_counter
);

END_PROGRAM

// ---- POUs/PRG_PMPS.TcPOU
PROGRAM PRG_PMPS
VAR
    fbArbiterIO : FB_SubSysToArbiter_IO;
END_VAR

g_FastFaultOutputK0.Execute(bAutoReset:=True);

g_FastFaultOutputK2.Execute(
    i_xVeto:= (  PMPS_GVL.stCurrentBeamParameters.aVetoDevices[PMPS.K_Stopper.MR1K1_OUT]
              ),
    bAutoReset:=TRUE
);

g_FastFaultOutputK3.Execute(
    i_xVeto:= TRUE,
    bAutoReset:=TRUE
);

(*
 ------ DISABLED UNTIL PMPS SIGNALS ARE RECEIVED ------

g_FastFaultOutputK3.Execute(
    i_xVeto:= (  PMPS_GVL.stCurrentBeamParameters.aStoppers[PMPS.K_Stopper.MR1K3_OUT]
                 OR PMPS_GVL.stCurrentBeamParameters.aStoppers[PMPS.K_Stopper.MR1K1_IN]
              ),
    bAutoReset:=TRUE
);
*)

g_FastFaultOutputK4.Execute(
    i_xVeto:= (  PMPS_GVL.stCurrentBeamParameters.aVetoDevices[PMPS.K_Stopper.MR1K1_IN]
                 OR PMPS_GVL.stCurrentBeamParameters.aVetoDevices[PMPS.K_Stopper.MR1K3_IN]
              ),
    bAutoReset:=TRUE
);

// Aggregate FastFaultOutputs into a single FastFault
g_FastFault(
    io_fbFFHWO := g_FastFaultOutputAll,
    i_xOK := (  g_FastFaultOutputK0.q_xFastFaultOut
                AND g_FastFaultOutputK2.q_xFastFaultOut
                AND g_FastFaultOutputK3.q_xFastFaultOut
                AND g_FastFaultOutputK4.q_xFastFaultOut
             ),
    i_xAutoReset:=TRUE
);

g_FastFaultOutputAll.Execute(bAutoReset:=True);

// Arbiter
g_fbArbiter1.AddRequest(nReqID := 42, stReqBp := PMPS_GVL.cstFullBeam, sDevName := 'plc-kfe-vac');
fbArbiterIO(Arbiter := g_fbArbiter1, fbFFHWO := g_FastFaultOutputK0);

END_PROGRAM

// ---- POUs/FB_EXT_TREATY_GAUGE.TcPOU
FUNCTION_BLOCK FB_EXT_TREATY_GAUGE
// Handle external gauge communicated to this PLC by a single dry-contact.
VAR_INPUT

    //	Setpoint agreed upon w/ the external system signified by the signal they send.
    rTREATY_SIGNAL_PRESS : REAL;

    // Presumed pressure if the signal is not received.
    rNO_SIGNAL_PRESS : REAL;
END_VAR
VAR_OUTPUT
    {attribute 'pytmc' := '
    pv:
    '}
    IG      : ST_VG;
    {attribute 'pytmc' := '
    pv:
    '}
    EXT_IG  : ST_EXT_GCC;
END_VAR
VAR

    // Input from AD's system indicating pressure belopw setpoint.
    i_xEXT_Press_OK AT %I* : BOOL;

END_VAR

EXT_IG.xIlk_Inp := i_xEXT_Press_OK;

IF i_xEXT_Press_OK = TRUE THEN
    IG.rPRESS := rTREATY_SIGNAL_PRESS;
    IG.xPRESS_OK := TRUE;
    IG.xAT_VAC := TRUE;
ELSE
    IG.rPRESS := rNO_SIGNAL_PRESS;
    IG.xPRESS_OK := FALSE;
    IG.xAT_VAC := FALSE;
END_IF

END_FUNCTION_BLOCK

// ---- POUs/FB_EXT_TREATY_VGC.TcPOU
FUNCTION_BLOCK FB_EXT_TREATY_VGC
VAR_INPUT
    TREATY_VGC : ST_VGC;
END_VAR
VAR_OUTPUT
END_VAR
VAR
    q_xTREATY_VGC_STATUS AT%Q*: BOOL;
END_VAR

q_xTREATY_VGC_STATUS := TREATY_VGC.eState = E_ValvePositionState.OPEN;

END_FUNCTION_BLOCK

// ---- POUs/FB_EXT_ILK.TcPOU
FUNCTION_BLOCK FB_EXT_ILK
VAR_INPUT
    VG	:	ST_VG;
END_VAR
VAR_IN_OUT
    ILK	:	ST_EXT_ILK;
END_VAR
VAR_OUTPUT
END_VAR
VAR
    q_xILK_OK_DO	 AT%Q*	:	BOOL; // Send the signal to indicate that the interlock pressure has been met.
END_VAR

// Indicate that the interlock condition is met.
ILK.xIlkOK 			:= (VG.rPRESS < ILK.rPRO_SP) AND (VG.xPRESS_OK);

// Raise the output signal if the interlock condition is met AND the signal is enabled.
q_xILK_OK_DO		:= (VG.rPRESS < ILK.rPRO_SP) AND (VG.xPRESS_OK) AND (ILK.xIlk_sw);

// Se PV  indicating the output status
ILK.q_xILK_OK_DO	:= q_xILK_OK_DO;

END_FUNCTION_BLOCK
